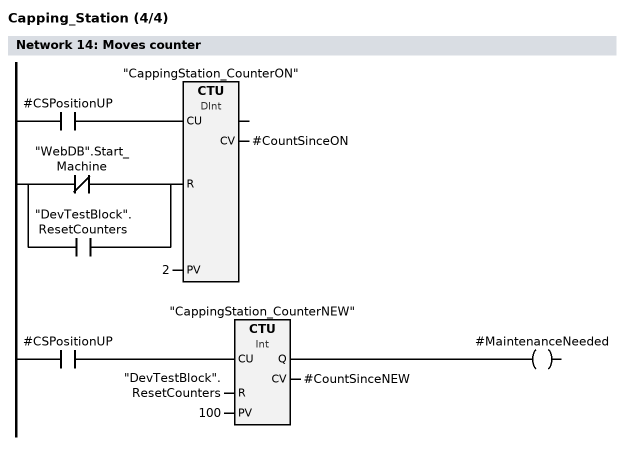
   RUNG wire#powerrail
      Contact( #CSPositionUP )
      { S7_Templates := "value_type := DInt" } "CappingStation_CounterON".CTU(r := wire#w1, pv := 2, cv => #CountSinceON)
   END_RUNG
   RUNG wire#powerrail
      I_Contact( "WebDB".Start_Machine )
   END_RUNG wire#w1
   RUNG wire#powerrail
      Contact( "DevTestBlock".ResetCounters )
   END_RUNG wire#w1
   RUNG wire#powerrail
      Contact( #CSPositionUP )
      { S7_Templates := "value_type := Int" } "CappingStation_CounterNEW".CTU(r := "DevTestBlock".ResetCounters, pv := 100, cv => #CountSinceNEW)
      Coil( #MaintenanceNeeded )
   END_RUNG
   // the same network as SCL:
   "CappingStation_CounterON".CTU(CU := #CSPositionUP,
                           R := NOT "WebDB".Start_Machine OR "DevTestBlock".ResetCounters,
                           PV := 2,
                           CV => #CountSinceON);
   "CappingStation_CounterNEW".CTU(CU := #CSPositionUP,
                           R := "DevTestBlock".ResetCounters,
                           PV := 100,
                           CV => #CountSinceNEW);
   #MaintenanceNeeded := "CappingStation_CounterNEW".Q;
END_REGION
END_FUNCTION_BLOCK

FUNCTION_BLOCK "Initial_Test_Squence"   // FB18, LAD
{ S7_Optimized_Access := 'TRUE' }
VERSION : 0.1
   VAR_INPUT
      ON : Bool;
      Position : DInt;
      HomingOK : Bool;
      InputTask : Bool;
      StepSizeInput : DInt := 100;
      AmountOfSteps : Int := 100;
   END_VAR
   VAR_OUTPUT
      StartMachine : Bool;
      StartHoming : Bool;
      StepSizeOutput : DInt := 1000;
      TestFinished : Bool;
      StartPosition : DInt;
      EndPositon : DInt;
   END_VAR
   VAR_IN_OUT
      StartTask : Bool;
   END_VAR
   VAR
      TurnOnM : Bool;
      StepNumber : Int;
      InternalWait : Bool;
      StepNumberNext : Int;
      ONM : Bool;
      TestFinishedM : Bool;
      StartTaskM : Bool;
   END_VAR
   VAR_TEMP   // added for the SCL form of the ladder/FBD networks
      _w1 : Bool;
   END_VAR
BEGIN

REGION Network 1: Turn On
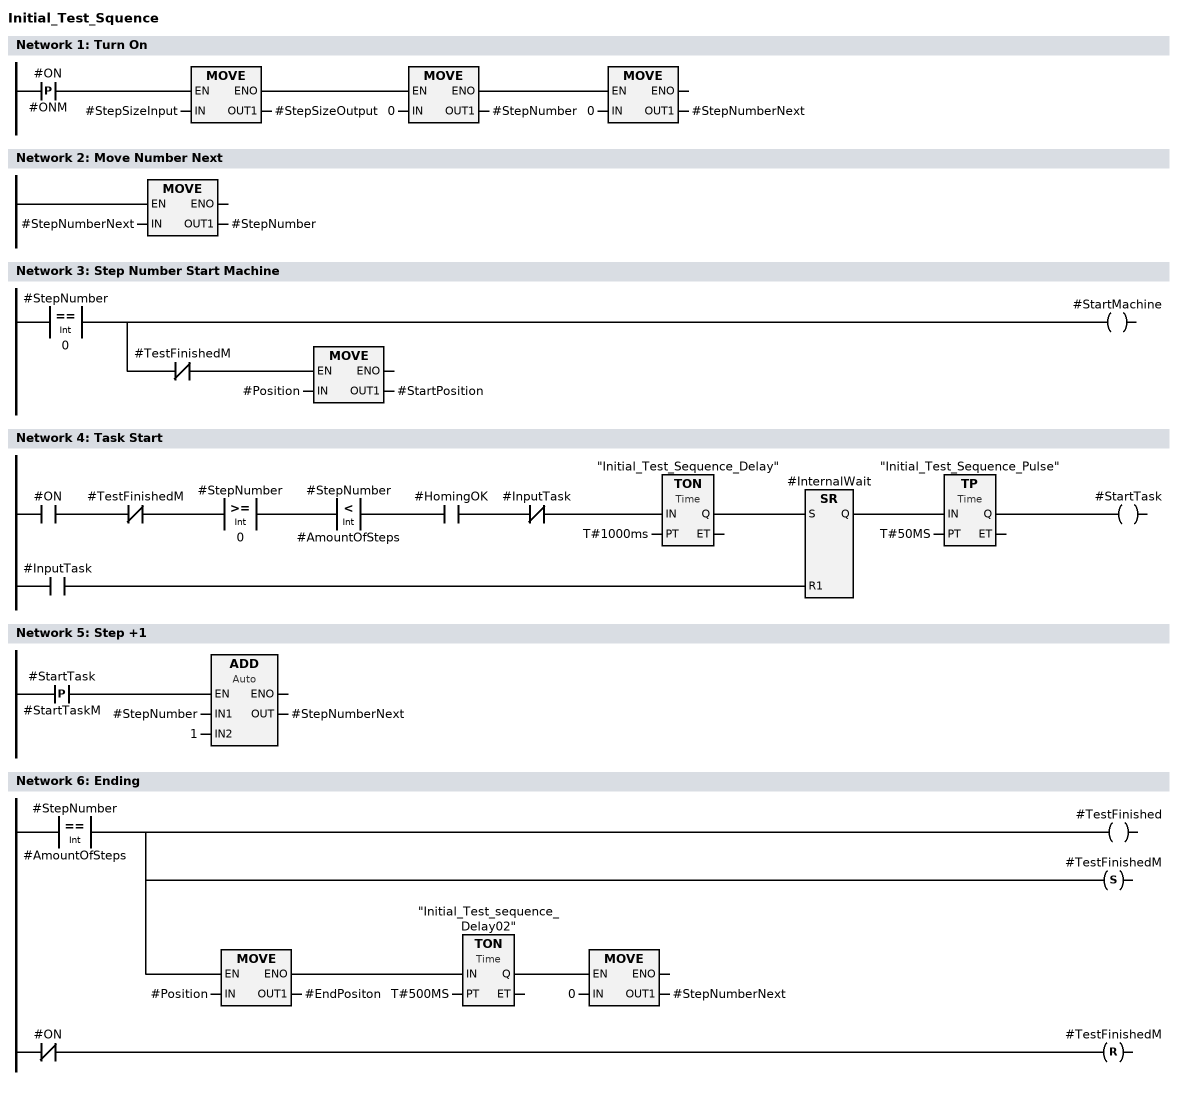
   RUNG wire#powerrail
      P_Contact(operand := #ON, bit := #ONM)
      Move(in := #StepSizeInput, out1 => #StepSizeOutput)
      Move(in := 0, out1 => #StepNumber)
      Move(in := 0, out1 => #StepNumberNext)
   END_RUNG
   // the same network as SCL:
   #_w1 := #ON AND NOT #ONM;   // rising edge of #ON
   #ONM := #ON;
   IF #_w1 THEN
       #StepSizeOutput := #StepSizeInput;
       #StepNumber := 0;
       #StepNumberNext := 0;
   END_IF;
END_REGION

REGION Network 2: Move Number Next
   RUNG wire#powerrail
      Move(in := #StepNumberNext, out1 => #StepNumber)
   END_RUNG
   // the same network as SCL:
   #StepNumber := #StepNumberNext;
END_REGION

REGION Network 3: Step Number Start Machine
   RUNG wire#powerrail
      { S7_Templates := "SrcType := Int" } EQ_Contact(in1 := #StepNumber, in2 := 0)
      wire#w1
      Coil( #StartMachine )
   END_RUNG
   RUNG wire#w1
      I_Contact( #TestFinishedM )
      Move(in := #Position, out1 => #StartPosition)
   END_RUNG
   // the same network as SCL:
   #StartMachine := #StepNumber = 0;
   IF #StartMachine AND NOT #TestFinishedM THEN #StartPosition := #Position; END_IF;
END_REGION

REGION Network 4: Task Start
   RUNG wire#powerrail
      Contact( #ON )
      I_Contact( #TestFinishedM )
      { S7_Templates := "SrcType := Int" } GE_Contact(in1 := #StepNumber, in2 := 0)
      { S7_Templates := "SrcType := Int" } LT_Contact(in1 := #StepNumber, in2 := #AmountOfSteps)
      Contact( #HomingOK )
      I_Contact( #InputTask )
      { S7_Templates := "time_type := Time" } "Initial_Test_Sequence_Delay".TON(pt := T#1000ms, et =>)
      S_SR(operand := #InternalWait, r1 := wire#w1)
      { S7_Templates := "time_type := Time" } "Initial_Test_Sequence_Pulse".TP(pt := T#50MS, et =>)
      Coil( #StartTask )
   END_RUNG
   RUNG wire#powerrail
      Contact( #InputTask )
   END_RUNG wire#w1
   // the same network as SCL:
   "Initial_Test_Sequence_Delay".TON(IN := #ON AND NOT #TestFinishedM AND (#StepNumber >= 0) AND (#StepNumber < #AmountOfSteps) AND #HomingOK AND NOT #InputTask,
                           PT := T#1000ms);
   IF "Initial_Test_Sequence_Delay".Q THEN
       #InternalWait := TRUE;   // SR flip-flop
   END_IF;
   IF #InputTask THEN #InternalWait := FALSE; END_IF;
   "Initial_Test_Sequence_Pulse".TP(IN := #InternalWait, PT := T#50MS);
   #StartTask := "Initial_Test_Sequence_Pulse".Q;
END_REGION

REGION Network 5: Step +1
   RUNG wire#powerrail
      P_Contact(operand := #StartTask, bit := #StartTaskM)
      Add(in1 := #StepNumber, in2 := 1, out => #StepNumberNext)
   END_RUNG
   // the same network as SCL:
   #_w1 := #StartTask AND NOT #StartTaskM;   // rising edge of #StartTask
   #StartTaskM := #StartTask;
   IF #_w1 THEN #StepNumberNext := #StepNumber + 1; END_IF;
END_REGION

REGION Network 6: Ending
   RUNG wire#powerrail
      { S7_Templates := "SrcType := Int" } EQ_Contact(in1 := #StepNumber, in2 := #AmountOfSteps)
      wire#w1
      Coil( #TestFinished )
   END_RUNG
   RUNG wire#w1
      S_Coil( #TestFinishedM )
   END_RUNG
   RUNG wire#w1
      Move(in := #Position, out1 => #EndPositon)
      { S7_Templates := "time_type := Time" } "Initial_Test_sequence_Delay02".TON(pt := T#500MS, et =>)
      Move(in := 0, out1 => #StepNumberNext)
   END_RUNG
   RUNG wire#powerrail
      I_Contact( #ON )
      R_Coil( #TestFinishedM )
   END_RUNG
   // the same network as SCL:
   #TestFinished := #StepNumber = #AmountOfSteps;
   IF #TestFinished THEN
       #TestFinishedM := TRUE;
       #EndPositon := #Position;
   END_IF;
   "Initial_Test_sequence_Delay02".TON(IN := #TestFinished, PT := T#500MS);
   IF "Initial_Test_sequence_Delay02".Q THEN #StepNumberNext := 0; END_IF;
   IF NOT #ON THEN #TestFinishedM := FALSE; END_IF;
END_REGION
END_FUNCTION_BLOCK

FUNCTION_BLOCK "UVLamp"   // FB19, LAD
TITLE = Description
{ S7_Optimized_Access := 'TRUE' }
VERSION : 0.1
// How to control and set the UV lamp:
// To control the lamp the machine needs to be started, all door closed and "LampFaultSignal" checked. After setting the setpoint 0-100 "LampSetpointInput" and enabling "LampEnable", the UV will work.
// 
// SafetyLimitSet - can be used to modify output range 
// 
// E-STOP - always check!
   VAR_INPUT
      Emergency : Bool;
      MachineStart : Bool;
      LampEnable : Bool;   // Device ready do use
      LampMode : Int;   // 0 by default
      LampSetpointInput : Real;   // Intensity %
      LampMaintenance : Int;   // N/A
      LampFaultSignal : Bool;   // Signal from the UV lamp
      DoorSensor : Bool;   // Connect direct
      XPosition : DInt;
      YPosition : DInt;
      WorkingRegionXstart : DInt;   // To be updated and connected to the UV lamp preferences in the MachineDB
      WorkingRegionXend : DInt := 500000;   // To be updated and connected to the UV lamp preferences in the MachineDB
      WorkingRegionYstart : DInt;   // To be updated and connected to the UV lamp preferences in the MachineDB
      WorkingRegionYend : DInt := 1500000;   // To be updated and connected to the UV lamp preferences in the MachineDB
      DevelopmentMode : Bool;
      FirstTurnOn : Bool;
   END_VAR
   VAR_OUTPUT
      LampEnabled : Bool;
      LampWorking : Bool;
      LampOutONOFF : Bool;
      LampDimming : UInt;
      LampIntensity : Real;   // Volts
      LampError : Bool;
      LampStatus : Int;   // N/A
   END_VAR
   VAR_IN_OUT
      LampInONOFF : Bool;   // Device use state
   END_VAR
   VAR
      InternalWorkingPermission : Bool;
      SetpointMax : UInt := 27648;   // 0 - 0V; 27648 - 10V;
      SetpointLimit : UInt := 27648;
      SetpointConversion : Real;
      SetpointOutput : UInt;
      SafetyLimitConversion : Real;
      IntensityConversion : Real;
   END_VAR
   VAR_TEMP
      WorkingRegionOK : Bool;
   END_VAR
   VAR CONSTANT
      SafetyLimitSet : Real := 60.0;   // 0-100%
   END_VAR
BEGIN

REGION Network 1: Working Region Check
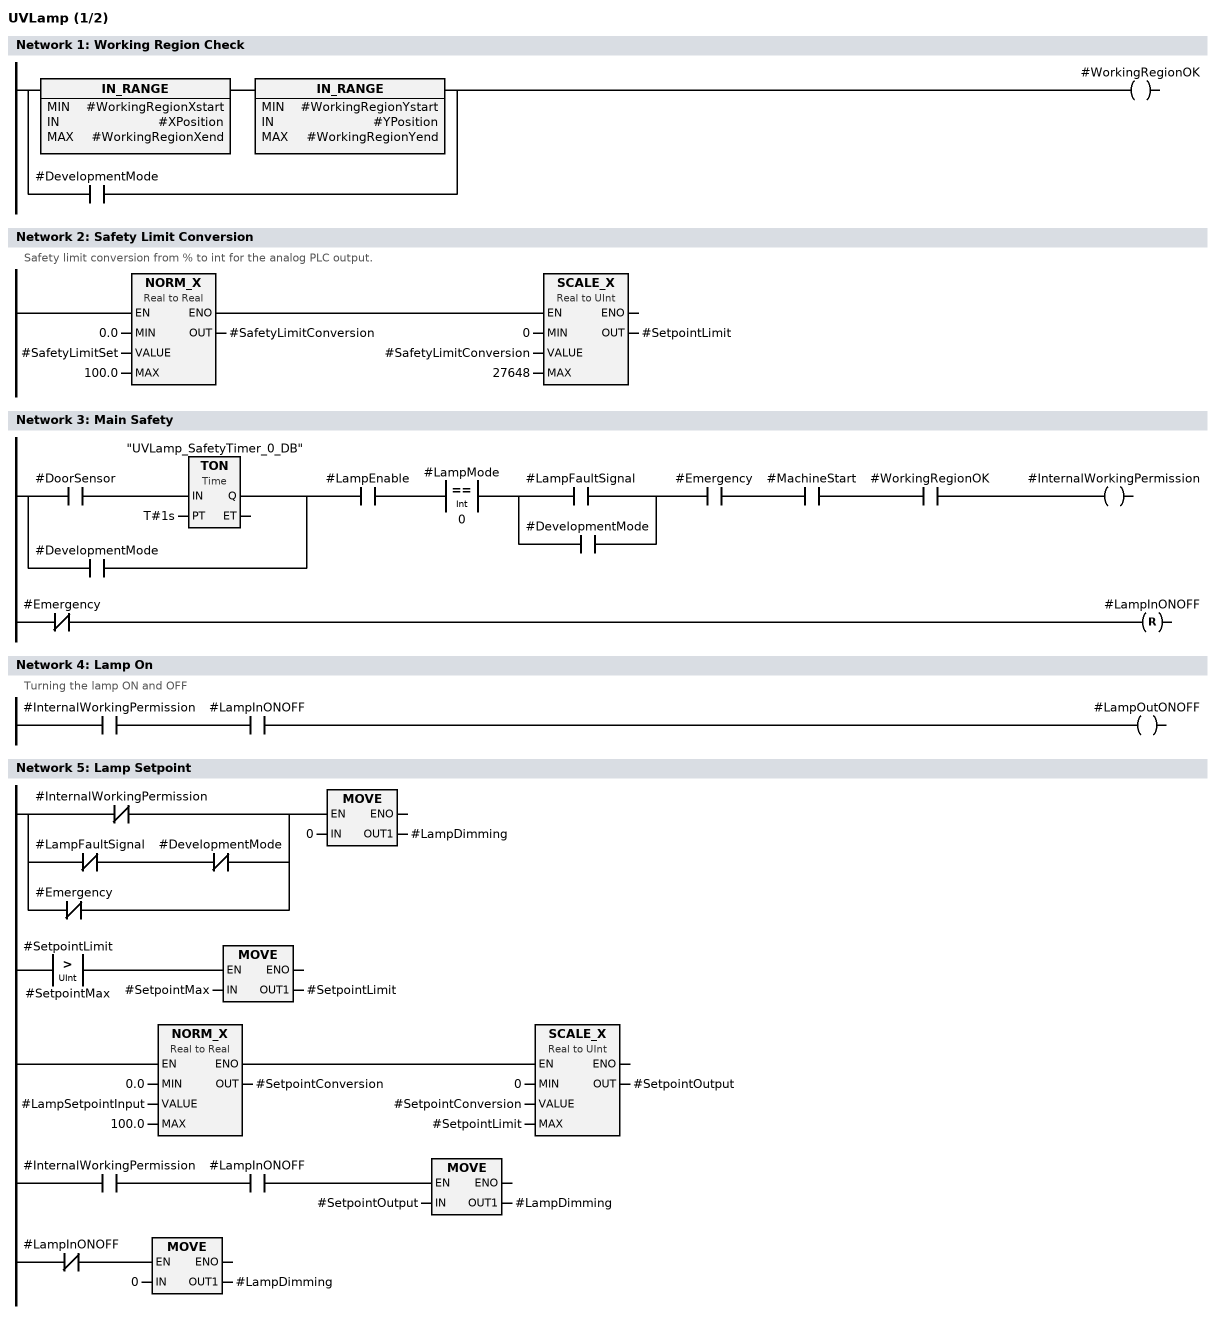
   RUNG wire#powerrail
      { S7_Templates := "SrcType := DInt" } InRange(min := #WorkingRegionXstart, in := #XPosition, max := #WorkingRegionXend)
      { S7_Templates := "SrcType := DInt" } InRange(min := #WorkingRegionYstart, in := #YPosition, max := #WorkingRegionYend)
      wire#w1
      Coil( #WorkingRegionOK )
   END_RUNG
   RUNG wire#powerrail
      Contact( #DevelopmentMode )
   END_RUNG wire#w1
   // the same network as SCL:
   #WorkingRegionOK := ((#WorkingRegionXstart <= #XPosition) AND (#XPosition <= #WorkingRegionXend) AND (#WorkingRegionYstart <= #YPosition) AND (#YPosition <= #WorkingRegionYend)) OR #DevelopmentMode;
END_REGION

REGION Network 2: Safety Limit Conversion
   // Safety limit conversion from % to int for the analog PLC output.
   RUNG wire#powerrail
      { S7_Templates := "[SrcType := Real, DestType := Real]" } Normalize(min := 0.0, value := #SafetyLimitSet, max := 100.0, out => #SafetyLimitConversion)
      { S7_Templates := "[SrcType := Real, DestType := UInt]" } Scale(min := 0, value := #SafetyLimitConversion, max := 27648, out => #SetpointLimit)
   END_RUNG
   // the same network as SCL:
   #SafetyLimitConversion := NORM_X(MIN := 0.0, VALUE := #SafetyLimitSet, MAX := 100.0);
   #SetpointLimit := SCALE_X(MIN := 0, VALUE := #SafetyLimitConversion, MAX := 27648);
END_REGION

REGION Network 3: Main Safety
   RUNG wire#powerrail
      Contact( #DoorSensor )
      { S7_Templates := "time_type := Time" } "UVLamp_SafetyTimer_0_DB".TON(pt := T#1s, et =>)
      wire#w1
      Contact( #LampEnable )
      { S7_Templates := "SrcType := Int" } EQ_Contact(in1 := #LampMode, in2 := 0)
      wire#w2
      Contact( #LampFaultSignal )
      wire#w3
      Contact( #Emergency )
      Contact( #MachineStart )
      Contact( #WorkingRegionOK )
      Coil( #InternalWorkingPermission )
   END_RUNG
   RUNG wire#powerrail
      Contact( #DevelopmentMode )
   END_RUNG wire#w1
   RUNG wire#w2
      Contact( #DevelopmentMode )
   END_RUNG wire#w3
   RUNG wire#powerrail
      I_Contact( #Emergency )
      R_Coil( #LampInONOFF )
   END_RUNG
   // the same network as SCL:
   "UVLamp_SafetyTimer_0_DB".TON(IN := #DoorSensor, PT := T#1s);
   #InternalWorkingPermission := ("UVLamp_SafetyTimer_0_DB".Q OR #DevelopmentMode) AND #LampEnable AND (#LampMode = 0) AND (#LampFaultSignal OR #DevelopmentMode) AND #Emergency AND #MachineStart AND #WorkingRegionOK;
   IF NOT #Emergency THEN #LampInONOFF := FALSE; END_IF;
END_REGION

REGION Network 4: Lamp On
   // Turning the lamp ON and OFF
   RUNG wire#powerrail
      Contact( #InternalWorkingPermission )
      Contact( #LampInONOFF )
      Coil( #LampOutONOFF )
   END_RUNG
   // the same network as SCL:
   #LampOutONOFF := #InternalWorkingPermission AND #LampInONOFF;
END_REGION

REGION Network 5: Lamp Setpoint
   RUNG wire#powerrail
      I_Contact( #InternalWorkingPermission )
      wire#w1
      Move(in := 0, out1 => #LampDimming)
   END_RUNG
   RUNG wire#powerrail
      I_Contact( #LampFaultSignal )
      I_Contact( #DevelopmentMode )
   END_RUNG wire#w1
   RUNG wire#powerrail
      I_Contact( #Emergency )
   END_RUNG wire#w1
   RUNG wire#powerrail
      { S7_Templates := "SrcType := UInt" } GT_Contact(in1 := #SetpointLimit, in2 := #SetpointMax)
      Move(in := #SetpointMax, out1 => #SetpointLimit)
   END_RUNG
   RUNG wire#powerrail
      { S7_Templates := "[SrcType := Real, DestType := Real]" } Normalize(min := 0.0, value := #LampSetpointInput, max := 100.0, out => #SetpointConversion)
      { S7_Templates := "[SrcType := Real, DestType := UInt]" } Scale(min := 0, value := #SetpointConversion, max := #SetpointLimit, out => #SetpointOutput)
   END_RUNG
   RUNG wire#powerrail
      Contact( #InternalWorkingPermission )
      Contact( #LampInONOFF )
      Move(in := #SetpointOutput, out1 => #LampDimming)
   END_RUNG
   RUNG wire#powerrail
      I_Contact( #LampInONOFF )
      Move(in := 0, out1 => #LampDimming)
   END_RUNG
   // the same network as SCL:
   IF NOT #InternalWorkingPermission OR (NOT #LampFaultSignal AND NOT #DevelopmentMode) OR NOT #Emergency THEN
       #LampDimming := 0;
   END_IF;
   IF #SetpointLimit > #SetpointMax THEN #SetpointLimit := #SetpointMax; END_IF;
   #SetpointConversion := NORM_X(MIN := 0.0, VALUE := #LampSetpointInput, MAX := 100.0);
   #SetpointOutput := SCALE_X(MIN := 0, VALUE := #SetpointConversion, MAX := #SetpointLimit);
   IF #InternalWorkingPermission AND #LampInONOFF THEN #LampDimming := #SetpointOutput; END_IF;
   IF NOT #LampInONOFF THEN #LampDimming := 0; END_IF;
END_REGION

REGION Network 6: Intensity Monitoring Conversion
   // Conversion of the intensity.
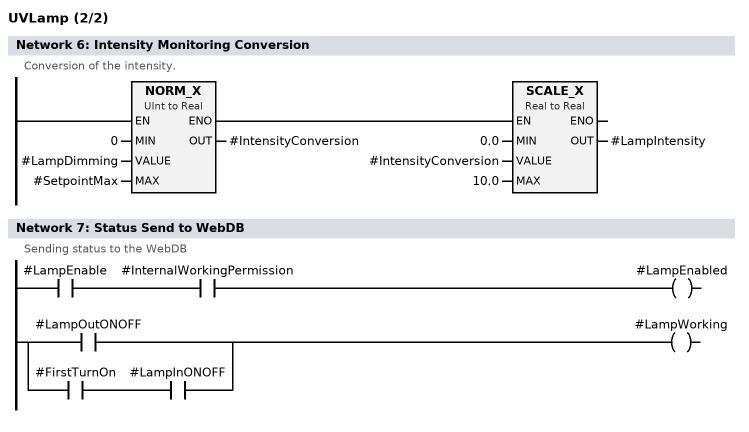
   RUNG wire#powerrail
      { S7_Templates := "[SrcType := UInt, DestType := Real]" } Normalize(min := 0, value := #LampDimming, max := #SetpointMax, out => #IntensityConversion)
      { S7_Templates := "[SrcType := Real, DestType := Real]" } Scale(min := 0.0, value := #IntensityConversion, max := 10.0, out => #LampIntensity)
   END_RUNG
   // the same network as SCL:
   #IntensityConversion := NORM_X(MIN := 0, VALUE := #LampDimming, MAX := #SetpointMax);
   #LampIntensity := SCALE_X(MIN := 0.0, VALUE := #IntensityConversion, MAX := 10.0);
END_REGION

REGION Network 7: Status Send to WebDB
   // Sending status to the WebDB
   RUNG wire#powerrail
      Contact( #LampEnable )
      Contact( #InternalWorkingPermission )
      Coil( #LampEnabled )
   END_RUNG
   RUNG wire#powerrail
      Contact( #LampOutONOFF )
      wire#w1
      Coil( #LampWorking )
   END_RUNG
   RUNG wire#powerrail
      Contact( #FirstTurnOn )
      Contact( #LampInONOFF )
   END_RUNG wire#w1
   // the same network as SCL:
   #LampEnabled := #LampEnable AND #InternalWorkingPermission;
   #LampWorking := #LampOutONOFF OR (#FirstTurnOn AND #LampInONOFF);
END_REGION
END_FUNCTION_BLOCK

FUNCTION_BLOCK "Stacklight"   // FB20, LAD
TITLE = Description:
{ S7_Optimized_Access := 'TRUE' }
VERSION : 0.1
// The stacklight is showing the status of the machine and checking different conditions:
// - errors from the drives (PLC)
// - communication (NOAH)
// - errors from the fluid supply (NOAH)
// - doors (PLC)
// 
// RED - default color, error or PLC is turning on
// ORANGE - door open or in maintenance mode
// GREEN - machine connected and working fine
// 
// RED-GREEN blinking - machine ready to connect
// 
// Date:
   VAR_INPUT
      Emergency : Bool;
      Mode : Int;
      RedIn : Bool;
      YellowIn : Bool;
      GreenIn : Bool;
      ReadyDevices : Bool;
      DoorOpen : Bool;
      Xvelocity : DInt;
      Yvelocity : DInt;
      MachineReadyPLC : Bool;
      MachineReadyNOAH : Bool;
      MachinePrintingPLC : Bool;
      MachinePrintingNOAH : Bool;
      MachineErrorPLC : Bool;
      MachineErrorNOAH : Bool;
      LED01 : Bool;
      LED02 : Bool;
      Maintenance : Int;
   END_VAR
   VAR_OUTPUT
      Status : Int;
      OutputColor : Int;
      StacklightCTRL01 : Bool;
      StacklightCTRL02 : Bool;
   END_VAR
   VAR_IN_OUT
      MachineConnectedNOAH : Bool;
   END_VAR
   VAR
      TriggerVelocityForMoving : DInt := 5;
      GreenInternal : Bool;
      YellowInternal : Bool;
      RedInternal : Bool;
      ColorInternal : Int;   // 0 = Red; 1 = Orange; 2 = Green;
      MachineMovingInternal : Bool;
      MachineConnectedPLC : Bool;
      MachineConnectedInternal : Bool;
   END_VAR
   VAR CONSTANT
      MachineConnectedWaitTime : Time := T#3s;
      MachineConnectedResetTime : Time := T#200ms;
   END_VAR
BEGIN

REGION Network 1: Machine Moving Status Read
   // Checking if the machine is moving.
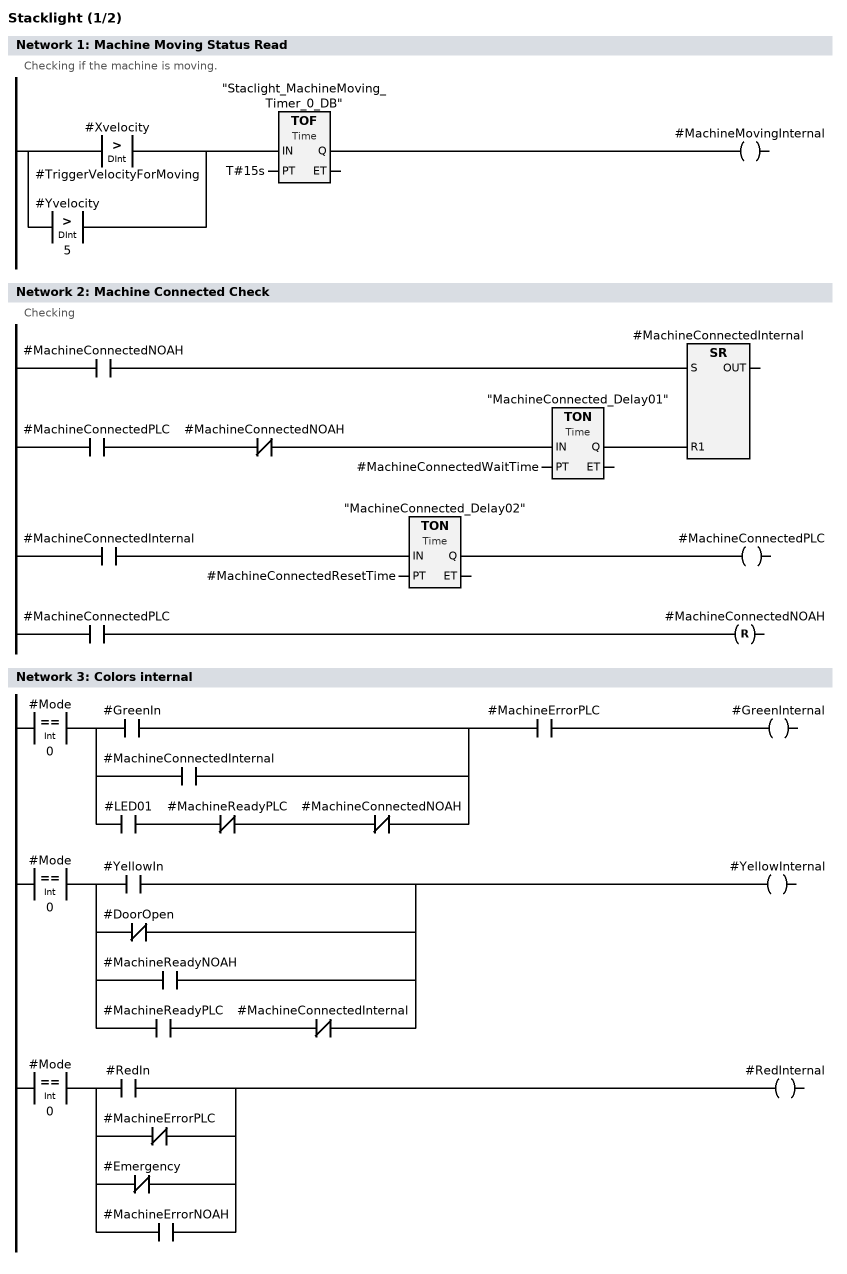
   RUNG wire#powerrail
      { S7_Templates := "SrcType := DInt" } GT_Contact(in1 := #Xvelocity, in2 := #TriggerVelocityForMoving)
      wire#w1
      { S7_Templates := "time_type := Time" } "Staclight_MachineMoving_Timer_0_DB".TOF(pt := T#15s, et =>)
      Coil( #MachineMovingInternal )
   END_RUNG
   RUNG wire#powerrail
      { S7_Templates := "SrcType := DInt" } GT_Contact(in1 := #Yvelocity, in2 := 5)
   END_RUNG wire#w1
   // the same network as SCL:
   "Staclight_MachineMoving_Timer_0_DB".TOF(IN := (#Xvelocity > #TriggerVelocityForMoving) OR (#Yvelocity > 5),
                           PT := T#15s);
   #MachineMovingInternal := "Staclight_MachineMoving_Timer_0_DB".Q;
END_REGION

REGION Network 2: Machine Connected Check
   // Checking
   RUNG wire#powerrail
      Contact( #MachineConnectedNOAH )
      S_SR(operand := #MachineConnectedInternal, r1 := wire#w1)
   END_RUNG
   RUNG wire#powerrail
      Contact( #MachineConnectedPLC )
      I_Contact( #MachineConnectedNOAH )
      { S7_Templates := "time_type := Time" } "MachineConnected_Delay01".TON(pt := #MachineConnectedWaitTime, et =>)
   END_RUNG wire#w1
   RUNG wire#powerrail
      Contact( #MachineConnectedInternal )
      { S7_Templates := "time_type := Time" } "MachineConnected_Delay02".TON(pt := #MachineConnectedResetTime, et =>)
      Coil( #MachineConnectedPLC )
   END_RUNG
   RUNG wire#powerrail
      Contact( #MachineConnectedPLC )
      R_Coil( #MachineConnectedNOAH )
   END_RUNG
   // the same network as SCL:
   "MachineConnected_Delay01".TON(IN := #MachineConnectedPLC AND NOT #MachineConnectedNOAH,
                           PT := #MachineConnectedWaitTime);
   IF #MachineConnectedNOAH THEN
       #MachineConnectedInternal := TRUE;   // SR flip-flop
   END_IF;
   IF "MachineConnected_Delay01".Q THEN #MachineConnectedInternal := FALSE; END_IF;
   "MachineConnected_Delay02".TON(IN := #MachineConnectedInternal, PT := #MachineConnectedResetTime);
   #MachineConnectedPLC := "MachineConnected_Delay02".Q;
   IF #MachineConnectedPLC THEN #MachineConnectedNOAH := FALSE; END_IF;
END_REGION

REGION Network 3: Colors internal
   RUNG wire#powerrail
      { S7_Templates := "SrcType := Int" } EQ_Contact(in1 := #Mode, in2 := 0)
      wire#w1
      Contact( #GreenIn )
      wire#w2
      Contact( #MachineErrorPLC )
      Coil( #GreenInternal )
   END_RUNG
   RUNG wire#w1
      Contact( #MachineConnectedInternal )
   END_RUNG wire#w2
   RUNG wire#w1
      Contact( #LED01 )
      I_Contact( #MachineReadyPLC )
      I_Contact( #MachineConnectedNOAH )
   END_RUNG wire#w2
   RUNG wire#powerrail
      { S7_Templates := "SrcType := Int" } EQ_Contact(in1 := #Mode, in2 := 0)
      wire#w3
      Contact( #YellowIn )
      wire#w4
      Coil( #YellowInternal )
   END_RUNG
   RUNG wire#w3
      I_Contact( #DoorOpen )
   END_RUNG wire#w4
   RUNG wire#w3
      Contact( #MachineReadyNOAH )
   END_RUNG wire#w4
   RUNG wire#w3
      Contact( #MachineReadyPLC )
      I_Contact( #MachineConnectedInternal )
   END_RUNG wire#w4
   RUNG wire#powerrail
      { S7_Templates := "SrcType := Int" } EQ_Contact(in1 := #Mode, in2 := 0)
      wire#w5
      Contact( #RedIn )
      wire#w6
      Coil( #RedInternal )
   END_RUNG
   RUNG wire#w5
      I_Contact( #MachineErrorPLC )
   END_RUNG wire#w6
   RUNG wire#w5
      I_Contact( #Emergency )
   END_RUNG wire#w6
   RUNG wire#w5
      Contact( #MachineErrorNOAH )
   END_RUNG wire#w6
   // the same network as SCL:
   #GreenInternal := (#Mode = 0) AND (#GreenIn OR #MachineConnectedInternal OR (#LED01 AND NOT #MachineReadyPLC AND NOT #MachineConnectedNOAH)) AND #MachineErrorPLC;
   #YellowInternal := (#Mode = 0) AND (#YellowIn OR NOT #DoorOpen OR #MachineReadyNOAH OR (#MachineReadyPLC AND NOT #MachineConnectedInternal));
   #RedInternal := (#Mode = 0) AND (#RedIn OR NOT #MachineErrorPLC OR NOT #Emergency OR #MachineErrorNOAH);
END_REGION

REGION Network 4: Status Move
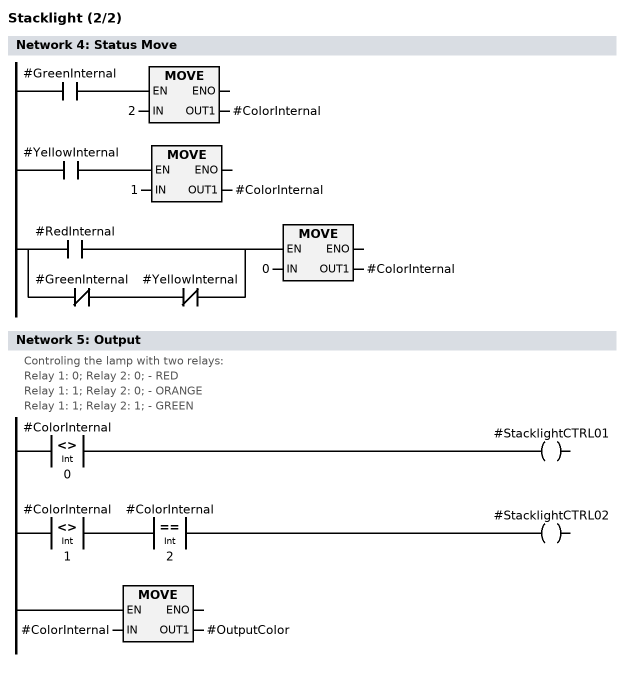
   RUNG wire#powerrail
      Contact( #GreenInternal )
      Move(in := 2, out1 => #ColorInternal)
   END_RUNG
   RUNG wire#powerrail
      Contact( #YellowInternal )
      Move(in := 1, out1 => #ColorInternal)
   END_RUNG
   RUNG wire#powerrail
      Contact( #RedInternal )
      wire#w1
      Move(in := 0, out1 => #ColorInternal)
   END_RUNG
   RUNG wire#powerrail
      I_Contact( #GreenInternal )
      I_Contact( #YellowInternal )
   END_RUNG wire#w1
   // the same network as SCL:
   IF #GreenInternal THEN #ColorInternal := 2; END_IF;
   IF #YellowInternal THEN #ColorInternal := 1; END_IF;
   IF #RedInternal OR (NOT #GreenInternal AND NOT #YellowInternal) THEN #ColorInternal := 0; END_IF;
END_REGION

REGION Network 5: Output
   // Controling the lamp with two relays:
   // Relay 1: 0; Relay 2: 0; - RED
   // Relay 1: 1; Relay 2: 0; - ORANGE
   // Relay 1: 1; Relay 2: 1; - GREEN
   RUNG wire#powerrail
      { S7_Templates := "SrcType := Int" } NE_Contact(in1 := #ColorInternal, in2 := 0)
      Coil( #StacklightCTRL01 )
   END_RUNG
   RUNG wire#powerrail
      { S7_Templates := "SrcType := Int" } NE_Contact(in1 := #ColorInternal, in2 := 1)
      { S7_Templates := "SrcType := Int" } EQ_Contact(in1 := #ColorInternal, in2 := 2)
      Coil( #StacklightCTRL02 )
   END_RUNG
   RUNG wire#powerrail
      Move(in := #ColorInternal, out1 => #OutputColor)
   END_RUNG
   // the same network as SCL:
   #StacklightCTRL01 := #ColorInternal <> 0;
   #StacklightCTRL02 := (#ColorInternal <> 1) AND (#ColorInternal = 2);
   #OutputColor := #ColorInternal;
END_REGION
END_FUNCTION_BLOCK

FUNCTION_BLOCK "Control_Buttons_Activation"   // FB23, LAD
{ S7_Optimized_Access := 'TRUE' }
VERSION : 0.1
   VAR_INPUT
      JogInZ1pos : Bool;
      JogInZ1neg : Bool;
      JogInZ2pos : Bool;
      JogInZ2neg : Bool;
   END_VAR
   VAR_OUTPUT
      Control_Buttons_Move_Permission : Bool;
      Control_Buttons_ActivatedOUT : Bool;
   END_VAR
   VAR
      Step01 : Bool;
      Step02 : Bool;
      Step03 : Bool;
      Step04 : Bool;
      Step05 : Bool;
      Step06 : Bool;
      Step07 : Bool;
      Step08 : Bool;
      AnyButtonPressed : Bool;
      AllButtonsPressed : Bool;
      ControlButtonsActivated : Bool;
   END_VAR
BEGIN

REGION Network 1: Any Button Pressed
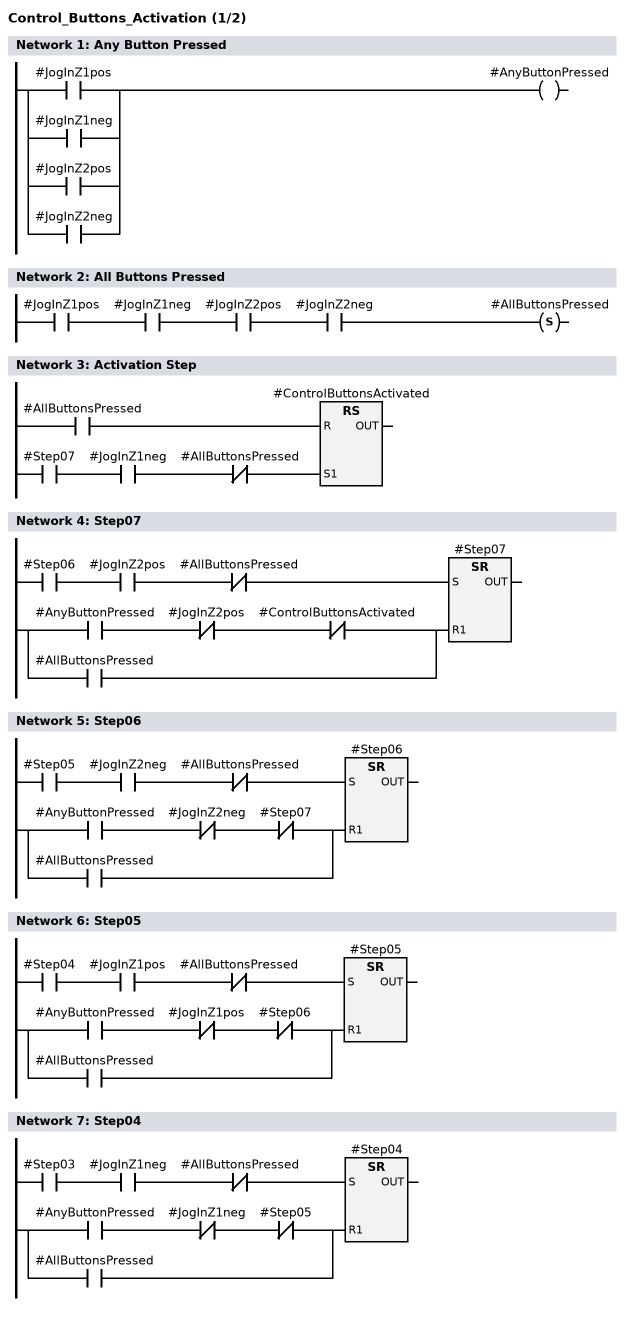
   RUNG wire#powerrail
      Contact( #JogInZ1pos )
      wire#w1
      Coil( #AnyButtonPressed )
   END_RUNG
   RUNG wire#powerrail
      Contact( #JogInZ1neg )
   END_RUNG wire#w1
   RUNG wire#powerrail
      Contact( #JogInZ2pos )
   END_RUNG wire#w1
   RUNG wire#powerrail
      Contact( #JogInZ2neg )
   END_RUNG wire#w1
   // the same network as SCL:
   #AnyButtonPressed := #JogInZ1pos OR #JogInZ1neg OR #JogInZ2pos OR #JogInZ2neg;
END_REGION

REGION Network 2: All Buttons Pressed
   RUNG wire#powerrail
      Contact( #JogInZ1pos )
      Contact( #JogInZ1neg )
      Contact( #JogInZ2pos )
      Contact( #JogInZ2neg )
      S_Coil( #AllButtonsPressed )
   END_RUNG
   // the same network as SCL:
   IF #JogInZ1pos AND #JogInZ1neg AND #JogInZ2pos AND #JogInZ2neg THEN #AllButtonsPressed := TRUE; END_IF;
END_REGION

REGION Network 3: Activation Step
   RUNG wire#powerrail
      Contact( #AllButtonsPressed )
      S_RS(operand := #ControlButtonsActivated, s1 := wire#w1)
   END_RUNG
   RUNG wire#powerrail
      Contact( #Step07 )
      Contact( #JogInZ1neg )
      I_Contact( #AllButtonsPressed )
   END_RUNG wire#w1
   // the same network as SCL:
   IF #AllButtonsPressed THEN
       #ControlButtonsActivated := FALSE;   // RS flip-flop
   END_IF;
   IF #Step07 AND #JogInZ1neg AND NOT #AllButtonsPressed THEN #ControlButtonsActivated := TRUE; END_IF;
END_REGION

REGION Network 4: Step07
   RUNG wire#powerrail
      Contact( #Step06 )
      Contact( #JogInZ2pos )
      I_Contact( #AllButtonsPressed )
      S_SR(operand := #Step07, r1 := wire#w1)
   END_RUNG
   RUNG wire#powerrail
      Contact( #AnyButtonPressed )
      I_Contact( #JogInZ2pos )
      I_Contact( #ControlButtonsActivated )
   END_RUNG wire#w1
   RUNG wire#powerrail
      Contact( #AllButtonsPressed )
   END_RUNG wire#w1
   // the same network as SCL:
   IF #Step06 AND #JogInZ2pos AND NOT #AllButtonsPressed THEN
       #Step07 := TRUE;   // SR flip-flop
   END_IF;
   IF (#AnyButtonPressed AND NOT #JogInZ2pos AND NOT #ControlButtonsActivated) OR #AllButtonsPressed THEN
       #Step07 := FALSE;
   END_IF;
END_REGION

REGION Network 5: Step06
   RUNG wire#powerrail
      Contact( #Step05 )
      Contact( #JogInZ2neg )
      I_Contact( #AllButtonsPressed )
      S_SR(operand := #Step06, r1 := wire#w1)
   END_RUNG
   RUNG wire#powerrail
      Contact( #AnyButtonPressed )
      I_Contact( #JogInZ2neg )
      I_Contact( #Step07 )
   END_RUNG wire#w1
   RUNG wire#powerrail
      Contact( #AllButtonsPressed )
   END_RUNG wire#w1
   // the same network as SCL:
   IF #Step05 AND #JogInZ2neg AND NOT #AllButtonsPressed THEN
       #Step06 := TRUE;   // SR flip-flop
   END_IF;
   IF (#AnyButtonPressed AND NOT #JogInZ2neg AND NOT #Step07) OR #AllButtonsPressed THEN
       #Step06 := FALSE;
   END_IF;
END_REGION

REGION Network 6: Step05
   RUNG wire#powerrail
      Contact( #Step04 )
      Contact( #JogInZ1pos )
      I_Contact( #AllButtonsPressed )
      S_SR(operand := #Step05, r1 := wire#w1)
   END_RUNG
   RUNG wire#powerrail
      Contact( #AnyButtonPressed )
      I_Contact( #JogInZ1pos )
      I_Contact( #Step06 )
   END_RUNG wire#w1
   RUNG wire#powerrail
      Contact( #AllButtonsPressed )
   END_RUNG wire#w1
   // the same network as SCL:
   IF #Step04 AND #JogInZ1pos AND NOT #AllButtonsPressed THEN
       #Step05 := TRUE;   // SR flip-flop
   END_IF;
   IF (#AnyButtonPressed AND NOT #JogInZ1pos AND NOT #Step06) OR #AllButtonsPressed THEN
       #Step05 := FALSE;
   END_IF;
END_REGION

REGION Network 7: Step04
   RUNG wire#powerrail
      Contact( #Step03 )
      Contact( #JogInZ1neg )
      I_Contact( #AllButtonsPressed )
      S_SR(operand := #Step04, r1 := wire#w1)
   END_RUNG
   RUNG wire#powerrail
      Contact( #AnyButtonPressed )
      I_Contact( #JogInZ1neg )
      I_Contact( #Step05 )
   END_RUNG wire#w1
   RUNG wire#powerrail
      Contact( #AllButtonsPressed )
   END_RUNG wire#w1
   // the same network as SCL:
   IF #Step03 AND #JogInZ1neg AND NOT #AllButtonsPressed THEN
       #Step04 := TRUE;   // SR flip-flop
   END_IF;
   IF (#AnyButtonPressed AND NOT #JogInZ1neg AND NOT #Step05) OR #AllButtonsPressed THEN
       #Step04 := FALSE;
   END_IF;
END_REGION

REGION Network 8: Step03
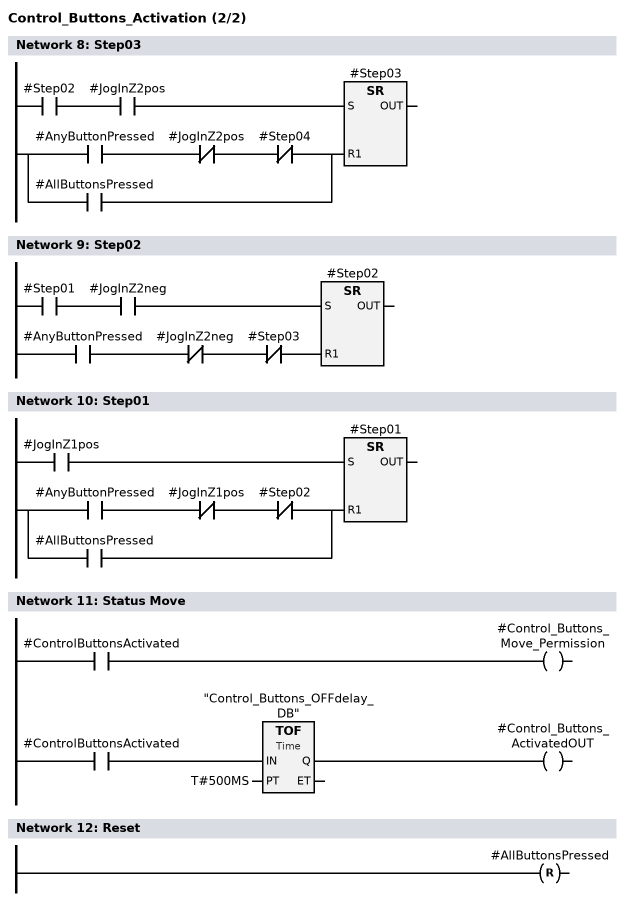
   RUNG wire#powerrail
      Contact( #Step02 )
      Contact( #JogInZ2pos )
      S_SR(operand := #Step03, r1 := wire#w1)
   END_RUNG
   RUNG wire#powerrail
      Contact( #AnyButtonPressed )
      I_Contact( #JogInZ2pos )
      I_Contact( #Step04 )
   END_RUNG wire#w1
   RUNG wire#powerrail
      Contact( #AllButtonsPressed )
   END_RUNG wire#w1
   // the same network as SCL:
   IF #Step02 AND #JogInZ2pos THEN
       #Step03 := TRUE;   // SR flip-flop
   END_IF;
   IF (#AnyButtonPressed AND NOT #JogInZ2pos AND NOT #Step04) OR #AllButtonsPressed THEN
       #Step03 := FALSE;
   END_IF;
END_REGION

REGION Network 9: Step02
   RUNG wire#powerrail
      Contact( #Step01 )
      Contact( #JogInZ2neg )
      S_SR(operand := #Step02, r1 := wire#w1)
   END_RUNG
   RUNG wire#powerrail
      Contact( #AnyButtonPressed )
      I_Contact( #JogInZ2neg )
      I_Contact( #Step03 )
   END_RUNG wire#w1
   // the same network as SCL:
   IF #Step01 AND #JogInZ2neg THEN
       #Step02 := TRUE;   // SR flip-flop
   END_IF;
   IF #AnyButtonPressed AND NOT #JogInZ2neg AND NOT #Step03 THEN #Step02 := FALSE; END_IF;
END_REGION

REGION Network 10: Step01
   RUNG wire#powerrail
      Contact( #JogInZ1pos )
      S_SR(operand := #Step01, r1 := wire#w1)
   END_RUNG
   RUNG wire#powerrail
      Contact( #AnyButtonPressed )
      I_Contact( #JogInZ1pos )
      I_Contact( #Step02 )
   END_RUNG wire#w1
   RUNG wire#powerrail
      Contact( #AllButtonsPressed )
   END_RUNG wire#w1
   // the same network as SCL:
   IF #JogInZ1pos THEN
       #Step01 := TRUE;   // SR flip-flop
   END_IF;
   IF (#AnyButtonPressed AND NOT #JogInZ1pos AND NOT #Step02) OR #AllButtonsPressed THEN
       #Step01 := FALSE;
   END_IF;
END_REGION

REGION Network 11: Status Move
   RUNG wire#powerrail
      Contact( #ControlButtonsActivated )
      Coil( #Control_Buttons_Move_Permission )
   END_RUNG
   RUNG wire#powerrail
      Contact( #ControlButtonsActivated )
      { S7_Templates := "time_type := Time" } "Control_Buttons_OFFdelay_DB".TOF(pt := T#500MS, et =>)
      Coil( #Control_Buttons_ActivatedOUT )
   END_RUNG
   // the same network as SCL:
   #Control_Buttons_Move_Permission := #ControlButtonsActivated;
   "Control_Buttons_OFFdelay_DB".TOF(IN := #ControlButtonsActivated, PT := T#500MS);
   #Control_Buttons_ActivatedOUT := "Control_Buttons_OFFdelay_DB".Q;
END_REGION

REGION Network 12: Reset
   RUNG wire#powerrail
      R_Coil( #AllButtonsPressed )
   END_RUNG
   // the same network as SCL:
   #AllButtonsPressed := FALSE;
END_REGION
END_FUNCTION_BLOCK

FUNCTION_BLOCK "Control_Buttons_Manipulate"   // FB24, LAD
{ S7_Optimized_Access := 'TRUE' }
VERSION : 0.1
// Simple control block to activate printhead motion in X and Y direction
   VAR_INPUT
      JogInZ1pos : Bool;
      JogInZ1neg : Bool;
      JogInZ2pos : Bool;
      JogInZ2neg : Bool;
      InXhome : Bool;
      InYhome : Bool;
      InZ1home : Bool;
      InZ2home : Bool;
      MovePermission : Bool;
      ReadyDevices : Bool;
   END_VAR
   VAR_OUTPUT
      JogOutXpos : Bool;
      JogOutXneg : Bool;
      JogOutYpos : Bool;
      JogOutYneg : Bool;
      JogOutZ1pos : Bool;
      JogOutZ1neg : Bool;
      JogOutZ2pos : Bool;
      JogOutZ2neg : Bool;
      XHoming : Bool;
      YHoming : Bool;
      Z1Homing : Bool;
      Z2Homing : Bool;
      StartMachine : Bool;
   END_VAR
   VAR
      ButtonsReadyToRead : Bool;
      XYmoveout : Bool;
   END_VAR
BEGIN

REGION Network 1: Start Machine
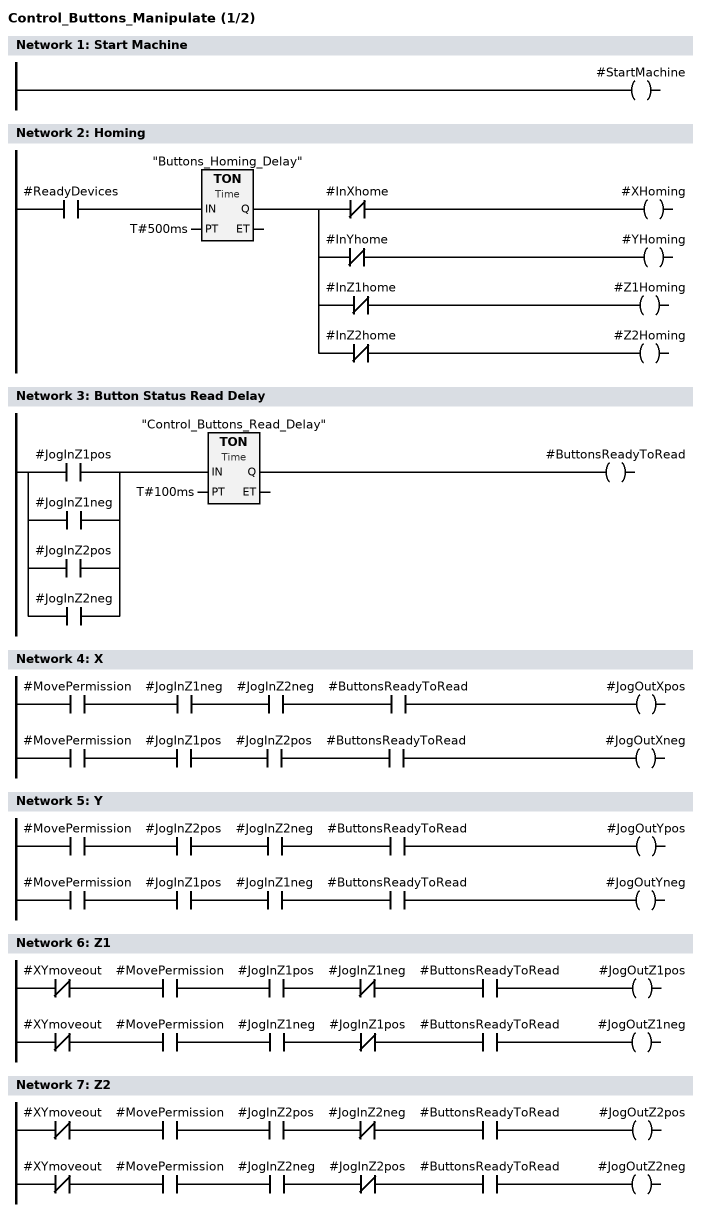
   RUNG wire#powerrail
      Coil( #StartMachine )
   END_RUNG
   // the same network as SCL:
   #StartMachine := TRUE;
END_REGION

REGION Network 2: Homing
   RUNG wire#powerrail
      Contact( #ReadyDevices )
      { S7_Templates := "time_type := Time" } "Buttons_Homing_Delay".TON(pt := T#500ms, et =>)
      wire#w1
      I_Contact( #InXhome )
      Coil( #XHoming )
   END_RUNG
   RUNG wire#w1
      I_Contact( #InYhome )
      Coil( #YHoming )
   END_RUNG
   RUNG wire#w1
      I_Contact( #InZ1home )
      Coil( #Z1Homing )
   END_RUNG
   RUNG wire#w1
      I_Contact( #InZ2home )
      Coil( #Z2Homing )
   END_RUNG
   // the same network as SCL:
   "Buttons_Homing_Delay".TON(IN := #ReadyDevices, PT := T#500ms);
   #XHoming := "Buttons_Homing_Delay".Q AND NOT #InXhome;
   #YHoming := "Buttons_Homing_Delay".Q AND NOT #InYhome;
   #Z1Homing := "Buttons_Homing_Delay".Q AND NOT #InZ1home;
   #Z2Homing := "Buttons_Homing_Delay".Q AND NOT #InZ2home;
END_REGION

REGION Network 3: Button Status Read Delay
   RUNG wire#powerrail
      Contact( #JogInZ1pos )
      wire#w1
      { S7_Templates := "time_type := Time" } "Control_Buttons_Read_Delay".TON(pt := T#100ms, et =>)
      Coil( #ButtonsReadyToRead )
   END_RUNG
   RUNG wire#powerrail
      Contact( #JogInZ1neg )
   END_RUNG wire#w1
   RUNG wire#powerrail
      Contact( #JogInZ2pos )
   END_RUNG wire#w1
   RUNG wire#powerrail
      Contact( #JogInZ2neg )
   END_RUNG wire#w1
   // the same network as SCL:
   "Control_Buttons_Read_Delay".TON(IN := #JogInZ1pos OR #JogInZ1neg OR #JogInZ2pos OR #JogInZ2neg,
                           PT := T#100ms);
   #ButtonsReadyToRead := "Control_Buttons_Read_Delay".Q;
END_REGION

REGION Network 4: X
   RUNG wire#powerrail
      Contact( #MovePermission )
      Contact( #JogInZ1neg )
      Contact( #JogInZ2neg )
      Contact( #ButtonsReadyToRead )
      Coil( #JogOutXpos )
   END_RUNG
   RUNG wire#powerrail
      Contact( #MovePermission )
      Contact( #JogInZ1pos )
      Contact( #JogInZ2pos )
      Contact( #ButtonsReadyToRead )
      Coil( #JogOutXneg )
   END_RUNG
   // the same network as SCL:
   #JogOutXpos := #MovePermission AND #JogInZ1neg AND #JogInZ2neg AND #ButtonsReadyToRead;
   #JogOutXneg := #MovePermission AND #JogInZ1pos AND #JogInZ2pos AND #ButtonsReadyToRead;
END_REGION

REGION Network 5: Y
   RUNG wire#powerrail
      Contact( #MovePermission )
      Contact( #JogInZ2pos )
      Contact( #JogInZ2neg )
      Contact( #ButtonsReadyToRead )
      Coil( #JogOutYpos )
   END_RUNG
   RUNG wire#powerrail
      Contact( #MovePermission )
      Contact( #JogInZ1pos )
      Contact( #JogInZ1neg )
      Contact( #ButtonsReadyToRead )
      Coil( #JogOutYneg )
   END_RUNG
   // the same network as SCL:
   #JogOutYpos := #MovePermission AND #JogInZ2pos AND #JogInZ2neg AND #ButtonsReadyToRead;
   #JogOutYneg := #MovePermission AND #JogInZ1pos AND #JogInZ1neg AND #ButtonsReadyToRead;
END_REGION

REGION Network 6: Z1
   RUNG wire#powerrail
      I_Contact( #XYmoveout )
      Contact( #MovePermission )
      Contact( #JogInZ1pos )
      I_Contact( #JogInZ1neg )
      Contact( #ButtonsReadyToRead )
      Coil( #JogOutZ1pos )
   END_RUNG
   RUNG wire#powerrail
      I_Contact( #XYmoveout )
      Contact( #MovePermission )
      Contact( #JogInZ1neg )
      I_Contact( #JogInZ1pos )
      Contact( #ButtonsReadyToRead )
      Coil( #JogOutZ1neg )
   END_RUNG
   // the same network as SCL:
   #JogOutZ1pos := NOT #XYmoveout AND #MovePermission AND #JogInZ1pos AND NOT #JogInZ1neg AND #ButtonsReadyToRead;
   #JogOutZ1neg := NOT #XYmoveout AND #MovePermission AND #JogInZ1neg AND NOT #JogInZ1pos AND #ButtonsReadyToRead;
END_REGION

REGION Network 7: Z2
   RUNG wire#powerrail
      I_Contact( #XYmoveout )
      Contact( #MovePermission )
      Contact( #JogInZ2pos )
      I_Contact( #JogInZ2neg )
      Contact( #ButtonsReadyToRead )
      Coil( #JogOutZ2pos )
   END_RUNG
   RUNG wire#powerrail
      I_Contact( #XYmoveout )
      Contact( #MovePermission )
      Contact( #JogInZ2neg )
      I_Contact( #JogInZ2pos )
      Contact( #ButtonsReadyToRead )
      Coil( #JogOutZ2neg )
   END_RUNG
   // the same network as SCL:
   #JogOutZ2pos := NOT #XYmoveout AND #MovePermission AND #JogInZ2pos AND NOT #JogInZ2neg AND #ButtonsReadyToRead;
   #JogOutZ2neg := NOT #XYmoveout AND #MovePermission AND #JogInZ2neg AND NOT #JogInZ2pos AND #ButtonsReadyToRead;
END_REGION

REGION Network 8: Status
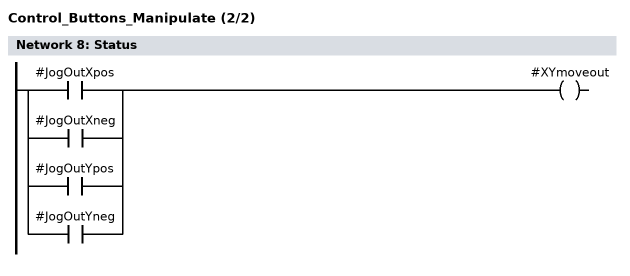
   RUNG wire#powerrail
      Contact( #JogOutXpos )
      wire#w1
      Coil( #XYmoveout )
   END_RUNG
   RUNG wire#powerrail
      Contact( #JogOutXneg )
   END_RUNG wire#w1
   RUNG wire#powerrail
      Contact( #JogOutYpos )
   END_RUNG wire#w1
   RUNG wire#powerrail
      Contact( #JogOutYneg )
   END_RUNG wire#w1
   // the same network as SCL:
   #XYmoveout := #JogOutXpos OR #JogOutXneg OR #JogOutYpos OR #JogOutYneg;
END_REGION
END_FUNCTION_BLOCK

FUNCTION_BLOCK "DataLogging"   // FB4, LAD
{ S7_Optimized_Access := 'TRUE' }
VERSION : 0.1
   VAR_INPUT
      CreateFile : Bool;
      StartLogging : Bool;
      Variable01in_Bool : Bool;
      Name_01 : String;
      Variable02in_Bool : Bool;
      Name_02 : String;
      Variable03in_Dint : DInt;
      Name_03 : String;
      Variable04in_Dint : DInt;
      Name_04 : String;
      Variable05in_Dint : DInt;
      Name_05 : String;
      Variable06in_Dint : DInt;
      Name_06 : String;
   END_VAR
   VAR_OUTPUT
      Variable01out_Bool : Bool;
      Variable02out_Bool : Bool;
      Variable03out_Dint : DInt;
      Variable04out_Dint : DInt;
      Variable05out_Dint : DInt;
      Variable06out_Dint : DInt;
      LogColumns : String;
   END_VAR
   VAR
      FileName : String := 'Logging_Test_01';
      REQ : Bool;
      ID : DWord;
      StartingTime : DTL;
      ReturnValue : Int;
      AmountOfRecords : UDInt := 10000;   // For 864000 and 10 records per sec = 24h
      StartLoggingM : Bool;
      WriteColumn : Int;
      Column01Internal : String;
      Column02Internal : String;
      Column03Internal : String;
      Column04Internal : String;
      Column05Internal : String;
      Column06Internal : String;
      WriteColumnReady : Bool;
      RecordCount : DInt;
   END_VAR
   VAR CONSTANT
      NameOfColumn01 : String := 'TestColumn_01';
      NameOfColumn02 : String := 'TestColumn_02';
   END_VAR
   VAR_TEMP   // added for the SCL form of the ladder/FBD networks
      _w1 : Bool;
      _w2 : Bool;
      _w3 : Bool;
      _w4 : Bool;
      _w5 : Bool;
   END_VAR
BEGIN

REGION Network 1: Start logging
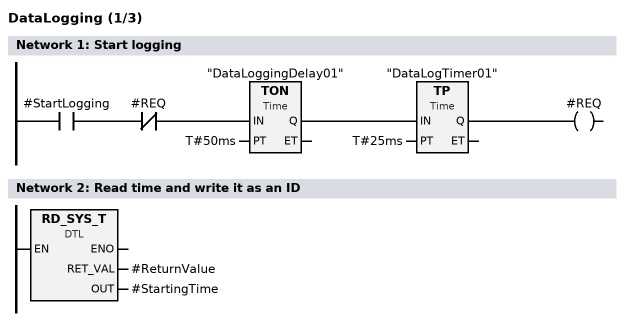
   RUNG wire#powerrail
      Contact( #StartLogging )
      I_Contact( #REQ )
      { S7_Templates := "time_type := Time" } "DataLoggingDelay01".TON(pt := T#50ms, et =>)
      { S7_Templates := "time_type := Time" } "DataLogTimer01".TP(pt := T#25ms, et =>)
      Coil( #REQ )
   END_RUNG
   // the same network as SCL:
   "DataLoggingDelay01".TON(IN := #StartLogging AND NOT #REQ, PT := T#50ms);
   "DataLogTimer01".TP(IN := "DataLoggingDelay01".Q, PT := T#25ms);
   #REQ := "DataLogTimer01".Q;
END_REGION

REGION Network 2: Read time and write it as an ID
   RUNG wire#powerrail
      { S7_Templates := "date_type := DTL" } RD_SYS_T(RET_VAL => #ReturnValue, OUT => #StartingTime)
   END_RUNG
   // the same network as SCL:
   #ReturnValue := RD_SYS_T(OUT => #StartingTime);
END_REGION

REGION Network 3: Write Column Names
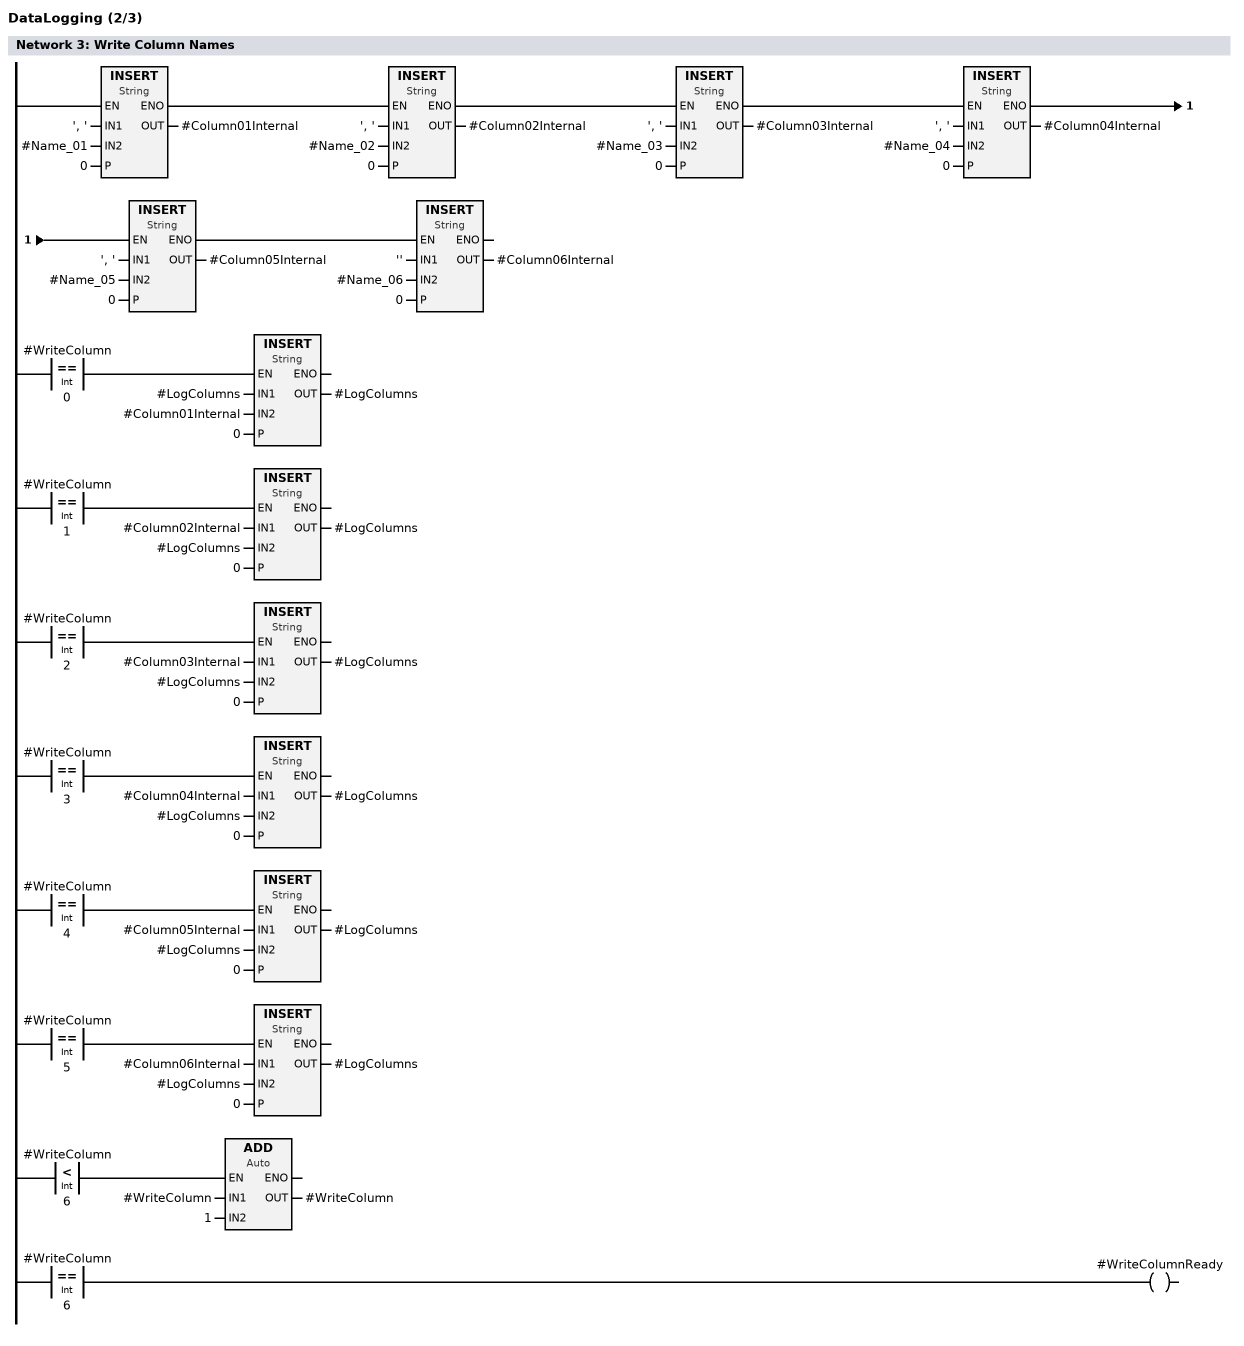
   RUNG wire#powerrail
      { S7_Templates := "str_type := String" } INSERT(IN1 := ', ', IN2 := #Name_01, P := 0, OUT => #Column01Internal)
      { S7_Templates := "str_type := String" } INSERT(IN1 := ', ', IN2 := #Name_02, P := 0, OUT => #Column02Internal)
      { S7_Templates := "str_type := String" } INSERT(IN1 := ', ', IN2 := #Name_03, P := 0, OUT => #Column03Internal)
      { S7_Templates := "str_type := String" } INSERT(IN1 := ', ', IN2 := #Name_04, P := 0, OUT => #Column04Internal)
      { S7_Templates := "str_type := String" } INSERT(IN1 := ', ', IN2 := #Name_05, P := 0, OUT => #Column05Internal)
      { S7_Templates := "str_type := String" } INSERT(IN1 := '', IN2 := #Name_06, P := 0, OUT => #Column06Internal)
   END_RUNG
   RUNG wire#powerrail
      { S7_Templates := "SrcType := Int" } EQ_Contact(in1 := #WriteColumn, in2 := 0)
      { S7_Templates := "str_type := String" } INSERT(IN1 := #LogColumns, IN2 := #Column01Internal, P := 0, OUT => #LogColumns)
   END_RUNG
   RUNG wire#powerrail
      { S7_Templates := "SrcType := Int" } EQ_Contact(in1 := #WriteColumn, in2 := 1)
      { S7_Templates := "str_type := String" } INSERT(IN1 := #Column02Internal, IN2 := #LogColumns, P := 0, OUT => #LogColumns)
   END_RUNG
   RUNG wire#powerrail
      { S7_Templates := "SrcType := Int" } EQ_Contact(in1 := #WriteColumn, in2 := 2)
      { S7_Templates := "str_type := String" } INSERT(IN1 := #Column03Internal, IN2 := #LogColumns, P := 0, OUT => #LogColumns)
   END_RUNG
   RUNG wire#powerrail
      { S7_Templates := "SrcType := Int" } EQ_Contact(in1 := #WriteColumn, in2 := 3)
      { S7_Templates := "str_type := String" } INSERT(IN1 := #Column04Internal, IN2 := #LogColumns, P := 0, OUT => #LogColumns)
   END_RUNG
   RUNG wire#powerrail
      { S7_Templates := "SrcType := Int" } EQ_Contact(in1 := #WriteColumn, in2 := 4)
      { S7_Templates := "str_type := String" } INSERT(IN1 := #Column05Internal, IN2 := #LogColumns, P := 0, OUT => #LogColumns)
   END_RUNG
   RUNG wire#powerrail
      { S7_Templates := "SrcType := Int" } EQ_Contact(in1 := #WriteColumn, in2 := 5)
      { S7_Templates := "str_type := String" } INSERT(IN1 := #Column06Internal, IN2 := #LogColumns, P := 0, OUT => #LogColumns)
   END_RUNG
   RUNG wire#powerrail
      { S7_Templates := "SrcType := Int" } LT_Contact(in1 := #WriteColumn, in2 := 6)
      Add(in1 := #WriteColumn, in2 := 1, out => #WriteColumn)
   END_RUNG
   RUNG wire#powerrail
      { S7_Templates := "SrcType := Int" } EQ_Contact(in1 := #WriteColumn, in2 := 6)
      Coil( #WriteColumnReady )
   END_RUNG
   // the same network as SCL:
   INSERT(IN1 := ', ', IN2 := #Name_01, P := 0, OUT => #Column01Internal, ENO => #_w1);
   INSERT(EN := #_w1, IN1 := ', ', IN2 := #Name_02, P := 0, OUT => #Column02Internal, ENO => #_w2);
   INSERT(EN := #_w2, IN1 := ', ', IN2 := #Name_03, P := 0, OUT => #Column03Internal, ENO => #_w3);
   INSERT(EN := #_w3, IN1 := ', ', IN2 := #Name_04, P := 0, OUT => #Column04Internal, ENO => #_w4);
   INSERT(EN := #_w4, IN1 := ', ', IN2 := #Name_05, P := 0, OUT => #Column05Internal, ENO => #_w5);
   IF #_w5 THEN INSERT(IN1 := '', IN2 := #Name_06, P := 0, OUT => #Column06Internal); END_IF;
   IF #WriteColumn = 0 THEN
       INSERT(IN1 := #LogColumns, IN2 := #Column01Internal, P := 0, OUT => #LogColumns);
   END_IF;
   IF #WriteColumn = 1 THEN
       INSERT(IN1 := #Column02Internal, IN2 := #LogColumns, P := 0, OUT => #LogColumns);
   END_IF;
   IF #WriteColumn = 2 THEN
       INSERT(IN1 := #Column03Internal, IN2 := #LogColumns, P := 0, OUT => #LogColumns);
   END_IF;
   IF #WriteColumn = 3 THEN
       INSERT(IN1 := #Column04Internal, IN2 := #LogColumns, P := 0, OUT => #LogColumns);
   END_IF;
   IF #WriteColumn = 4 THEN
       INSERT(IN1 := #Column05Internal, IN2 := #LogColumns, P := 0, OUT => #LogColumns);
   END_IF;
   IF #WriteColumn = 5 THEN
       INSERT(IN1 := #Column06Internal, IN2 := #LogColumns, P := 0, OUT => #LogColumns);
   END_IF;
   IF #WriteColumn < 6 THEN #WriteColumn := #WriteColumn + 1; END_IF;
   #WriteColumnReady := #WriteColumn = 6;
END_REGION

REGION Network 4: Data Logging Transfer
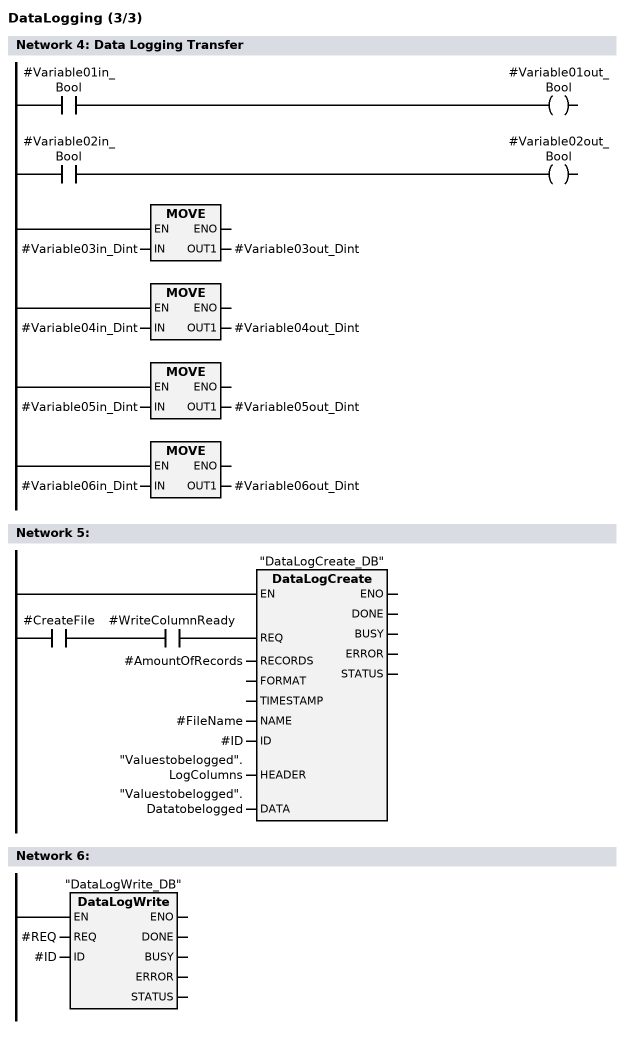
   RUNG wire#powerrail
      Contact( #Variable01in_Bool )
      Coil( #Variable01out_Bool )
   END_RUNG
   RUNG wire#powerrail
      Contact( #Variable02in_Bool )
      Coil( #Variable02out_Bool )
   END_RUNG
   RUNG wire#powerrail
      Move(in := #Variable03in_Dint, out1 => #Variable03out_Dint)
   END_RUNG
   RUNG wire#powerrail
      Move(in := #Variable04in_Dint, out1 => #Variable04out_Dint)
   END_RUNG
   RUNG wire#powerrail
      Move(in := #Variable05in_Dint, out1 => #Variable05out_Dint)
   END_RUNG
   RUNG wire#powerrail
      Move(in := #Variable06in_Dint, out1 => #Variable06out_Dint)
   END_RUNG
   // the same network as SCL:
   #Variable01out_Bool := #Variable01in_Bool;
   #Variable02out_Bool := #Variable02in_Bool;
   #Variable03out_Dint := #Variable03in_Dint;
   #Variable04out_Dint := #Variable04in_Dint;
   #Variable05out_Dint := #Variable05in_Dint;
   #Variable06out_Dint := #Variable06in_Dint;
END_REGION

REGION Network 5
   RUNG wire#powerrail
      "DataLogCreate_DB".DataLogCreate(REQ := wire#w1, RECORDS := #AmountOfRecords, FORMAT :=, TIMESTAMP :=, "NAME" := #FileName, ID := #ID, HEADER := "Valuestobelogged".LogColumns, DATA := "Valuestobelogged".Datatobelogged, DONE =>, BUSY =>, ERROR =>, STATUS =>)
   END_RUNG
   RUNG wire#powerrail
      Contact( #CreateFile )
      Contact( #WriteColumnReady )
   END_RUNG wire#w1
   // the same network as SCL:
   "DataLogCreate_DB"(REQ := #CreateFile AND #WriteColumnReady,   // DataLogCreate
                      RECORDS := #AmountOfRecords,
                      "NAME" := #FileName,
                      ID := #ID,
                      HEADER := "Valuestobelogged".LogColumns,
                      DATA := "Valuestobelogged".Datatobelogged);
END_REGION

REGION Network 6
   RUNG wire#powerrail
      "DataLogWrite_DB".DataLogWrite(REQ := #REQ, ID := #ID, DONE =>, BUSY =>, ERROR =>, STATUS =>)
   END_RUNG
   // the same network as SCL:
   "DataLogWrite_DB"(REQ := #REQ, ID := #ID);   // DataLogWrite
END_REGION
END_FUNCTION_BLOCK

FUNCTION_BLOCK "ZAxis_RelativeMotion_Test"   // FB25, LAD
{ S7_Optimized_Access := 'TRUE' }
VERSION : 0.1
   VAR_INPUT
      StartTest : Bool;
      EndTest : Bool;
      AmountOfSteps : DInt := 3000;
      StepSizeInput : DInt := 100;
      Position : DInt := 0;
      AxisMoving : Bool;
   END_VAR
   VAR_OUTPUT
      StartTask : Bool;
      StepSize : DInt;
      StepNumber : DInt;
      CreateLogFile : Bool;
      StartLog : Bool;
      Comment : String;
   END_VAR
   VAR
      TestActiveInternal : Bool;
      ActualStep : DInt := 9999;
      StepCountNext : DInt := 1;
      MovingInternal : Bool;
      ChangingCount : Bool;
      StartTaskM : Bool;
      LogCreatingReady : Bool;
   END_VAR
BEGIN

REGION Network 1: Log Creating
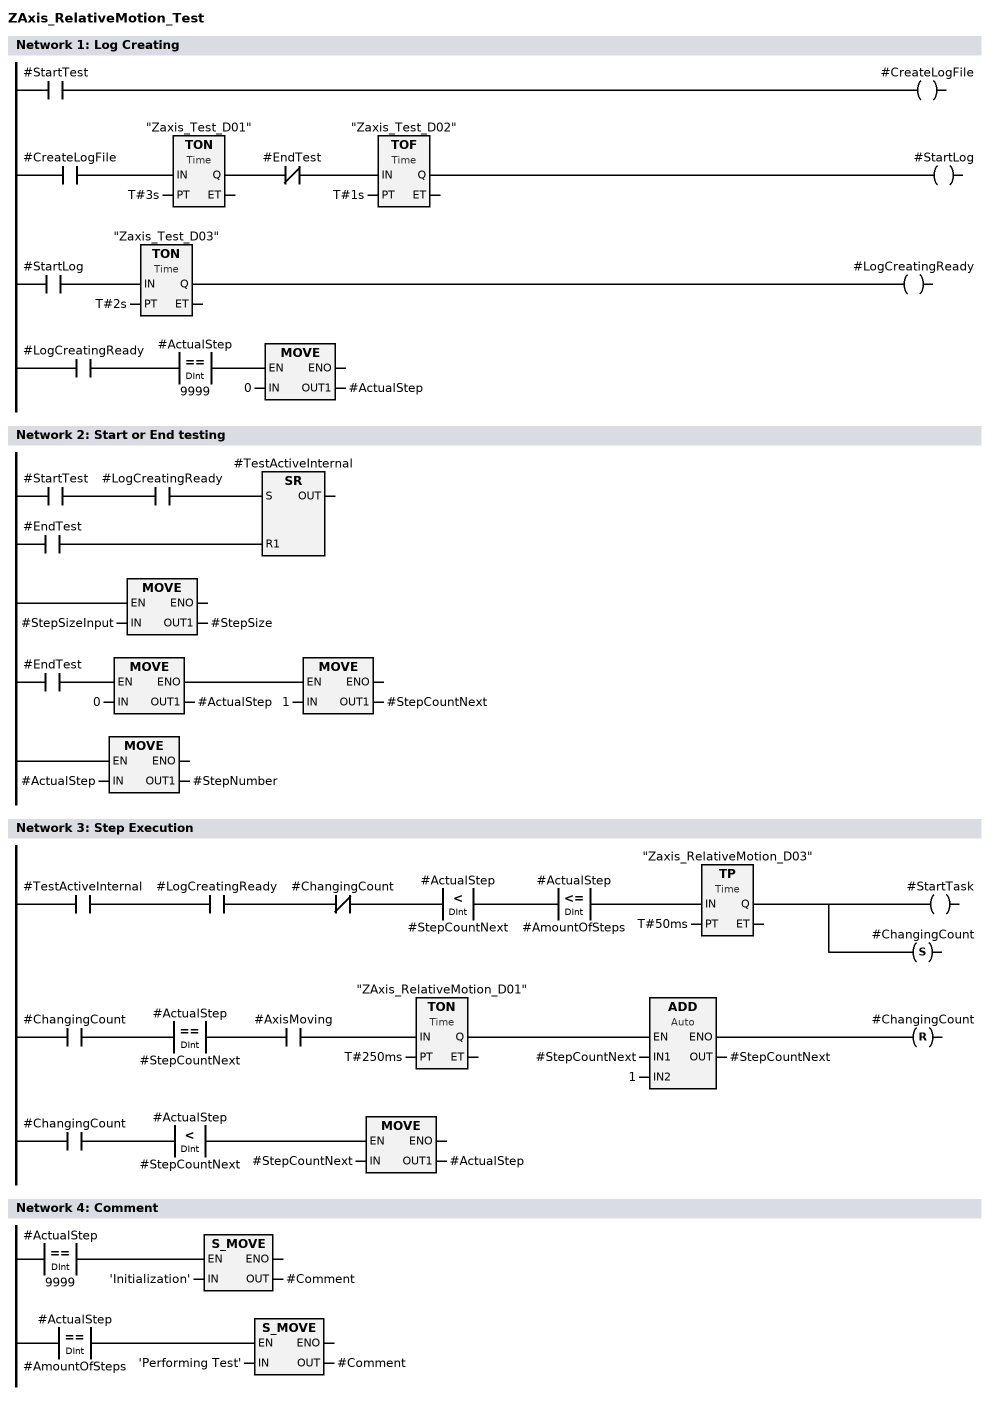
   RUNG wire#powerrail
      Contact( #StartTest )
      Coil( #CreateLogFile )
   END_RUNG
   RUNG wire#powerrail
      Contact( #CreateLogFile )
      { S7_Templates := "time_type := Time" } "Zaxis_Test_D01".TON(pt := T#3s, et =>)
      I_Contact( #EndTest )
      { S7_Templates := "time_type := Time" } "Zaxis_Test_D02".TOF(pt := T#1s, et =>)
      Coil( #StartLog )
   END_RUNG
   RUNG wire#powerrail
      Contact( #StartLog )
      { S7_Templates := "time_type := Time" } "Zaxis_Test_D03".TON(pt := T#2s, et =>)
      Coil( #LogCreatingReady )
   END_RUNG
   RUNG wire#powerrail
      Contact( #LogCreatingReady )
      { S7_Templates := "SrcType := DInt" } EQ_Contact(in1 := #ActualStep, in2 := 9999)
      Move(in := 0, out1 => #ActualStep)
   END_RUNG
   // the same network as SCL:
   #CreateLogFile := #StartTest;
   "Zaxis_Test_D01".TON(IN := #CreateLogFile, PT := T#3s);
   "Zaxis_Test_D02".TOF(IN := "Zaxis_Test_D01".Q AND NOT #EndTest, PT := T#1s);
   #StartLog := "Zaxis_Test_D02".Q;
   "Zaxis_Test_D03".TON(IN := #StartLog, PT := T#2s);
   #LogCreatingReady := "Zaxis_Test_D03".Q;
   IF #LogCreatingReady AND (#ActualStep = 9999) THEN #ActualStep := 0; END_IF;
END_REGION

REGION Network 2: Start or End testing
   RUNG wire#powerrail
      Contact( #StartTest )
      Contact( #LogCreatingReady )
      S_SR(operand := #TestActiveInternal, r1 := wire#w1)
   END_RUNG
   RUNG wire#powerrail
      Contact( #EndTest )
   END_RUNG wire#w1
   RUNG wire#powerrail
      Move(in := #StepSizeInput, out1 => #StepSize)
   END_RUNG
   RUNG wire#powerrail
      Contact( #EndTest )
      Move(in := 0, out1 => #ActualStep)
      Move(in := 1, out1 => #StepCountNext)
   END_RUNG
   RUNG wire#powerrail
      Move(in := #ActualStep, out1 => #StepNumber)
   END_RUNG
   // the same network as SCL:
   IF #StartTest AND #LogCreatingReady THEN
       #TestActiveInternal := TRUE;   // SR flip-flop
   END_IF;
   IF #EndTest THEN #TestActiveInternal := FALSE; END_IF;
   #StepSize := #StepSizeInput;
   IF #EndTest THEN
       #ActualStep := 0;
       #StepCountNext := 1;
   END_IF;
   #StepNumber := #ActualStep;
END_REGION

REGION Network 3: Step Execution
   RUNG wire#powerrail
      Contact( #TestActiveInternal )
      Contact( #LogCreatingReady )
      I_Contact( #ChangingCount )
      { S7_Templates := "SrcType := DInt" } LT_Contact(in1 := #ActualStep, in2 := #StepCountNext)
      { S7_Templates := "SrcType := DInt" } LE_Contact(in1 := #ActualStep, in2 := #AmountOfSteps)
      { S7_Templates := "time_type := Time" } "Zaxis_RelativeMotion_D03".TP(pt := T#50ms, et =>)
      wire#w1
      Coil( #StartTask )
   END_RUNG
   RUNG wire#w1
      S_Coil( #ChangingCount )
   END_RUNG
   RUNG wire#powerrail
      Contact( #ChangingCount )
      { S7_Templates := "SrcType := DInt" } EQ_Contact(in1 := #ActualStep, in2 := #StepCountNext)
      Contact( #AxisMoving )
      { S7_Templates := "time_type := Time" } "ZAxis_RelativeMotion_D01".TON(pt := T#250ms, et =>)
      Add(in1 := #StepCountNext, in2 := 1, out => #StepCountNext)
      R_Coil( #ChangingCount )
   END_RUNG
   RUNG wire#powerrail
      Contact( #ChangingCount )
      { S7_Templates := "SrcType := DInt" } LT_Contact(in1 := #ActualStep, in2 := #StepCountNext)
      Move(in := #StepCountNext, out1 => #ActualStep)
   END_RUNG
   // the same network as SCL:
   "Zaxis_RelativeMotion_D03".TP(IN := #TestActiveInternal AND #LogCreatingReady AND NOT #ChangingCount AND (#ActualStep < #StepCountNext) AND (#ActualStep <= #AmountOfSteps),
                           PT := T#50ms);
   #StartTask := "Zaxis_RelativeMotion_D03".Q;
   IF "Zaxis_RelativeMotion_D03".Q THEN #ChangingCount := TRUE; END_IF;
   "ZAxis_RelativeMotion_D01".TON(IN := #ChangingCount AND (#ActualStep = #StepCountNext) AND #AxisMoving,
                           PT := T#250ms);
   IF "ZAxis_RelativeMotion_D01".Q THEN
       #StepCountNext := #StepCountNext + 1;
       #ChangingCount := FALSE;
   END_IF;
   IF #ChangingCount AND (#ActualStep < #StepCountNext) THEN #ActualStep := #StepCountNext; END_IF;
END_REGION

REGION Network 4: Comment
   RUNG wire#powerrail
      { S7_Templates := "SrcType := DInt" } EQ_Contact(in1 := #ActualStep, in2 := 9999)
      S_Move(in := 'Initialization', out => #Comment)
   END_RUNG
   RUNG wire#powerrail
      { S7_Templates := "SrcType := DInt" } EQ_Contact(in1 := #ActualStep, in2 := #AmountOfSteps)
      S_Move(in := 'Performing Test', out => #Comment)
   END_RUNG
   // the same network as SCL:
   IF #ActualStep = 9999 THEN #Comment := 'Initialization'; END_IF;
   IF #ActualStep = #AmountOfSteps THEN #Comment := 'Performing Test'; END_IF;
END_REGION
END_FUNCTION_BLOCK

ORGANIZATION_BLOCK "Work Cyclic"   // OB30, LAD, CyclicInterrupt
TITLE = Description:
{ S7_Optimized_Access := 'TRUE' }
VERSION : 0.1
// Operations that are supposed to be executed in a precise cycle time, which is temporary set to 45ms. It is important to connect this time with the read/write time of the WebDB (NOAH).
   VAR_INPUT
      Initial_Call : Bool;   // Initial call of this OB
      Event_Count : Int;   // Events discarded
   END_VAR
   VAR_TEMP   // added for the SCL form of the ladder/FBD networks
      _w1 : Bool;
   END_VAR
BEGIN

REGION Network 1: AXIS Z1 Control CMMT V2 To Update
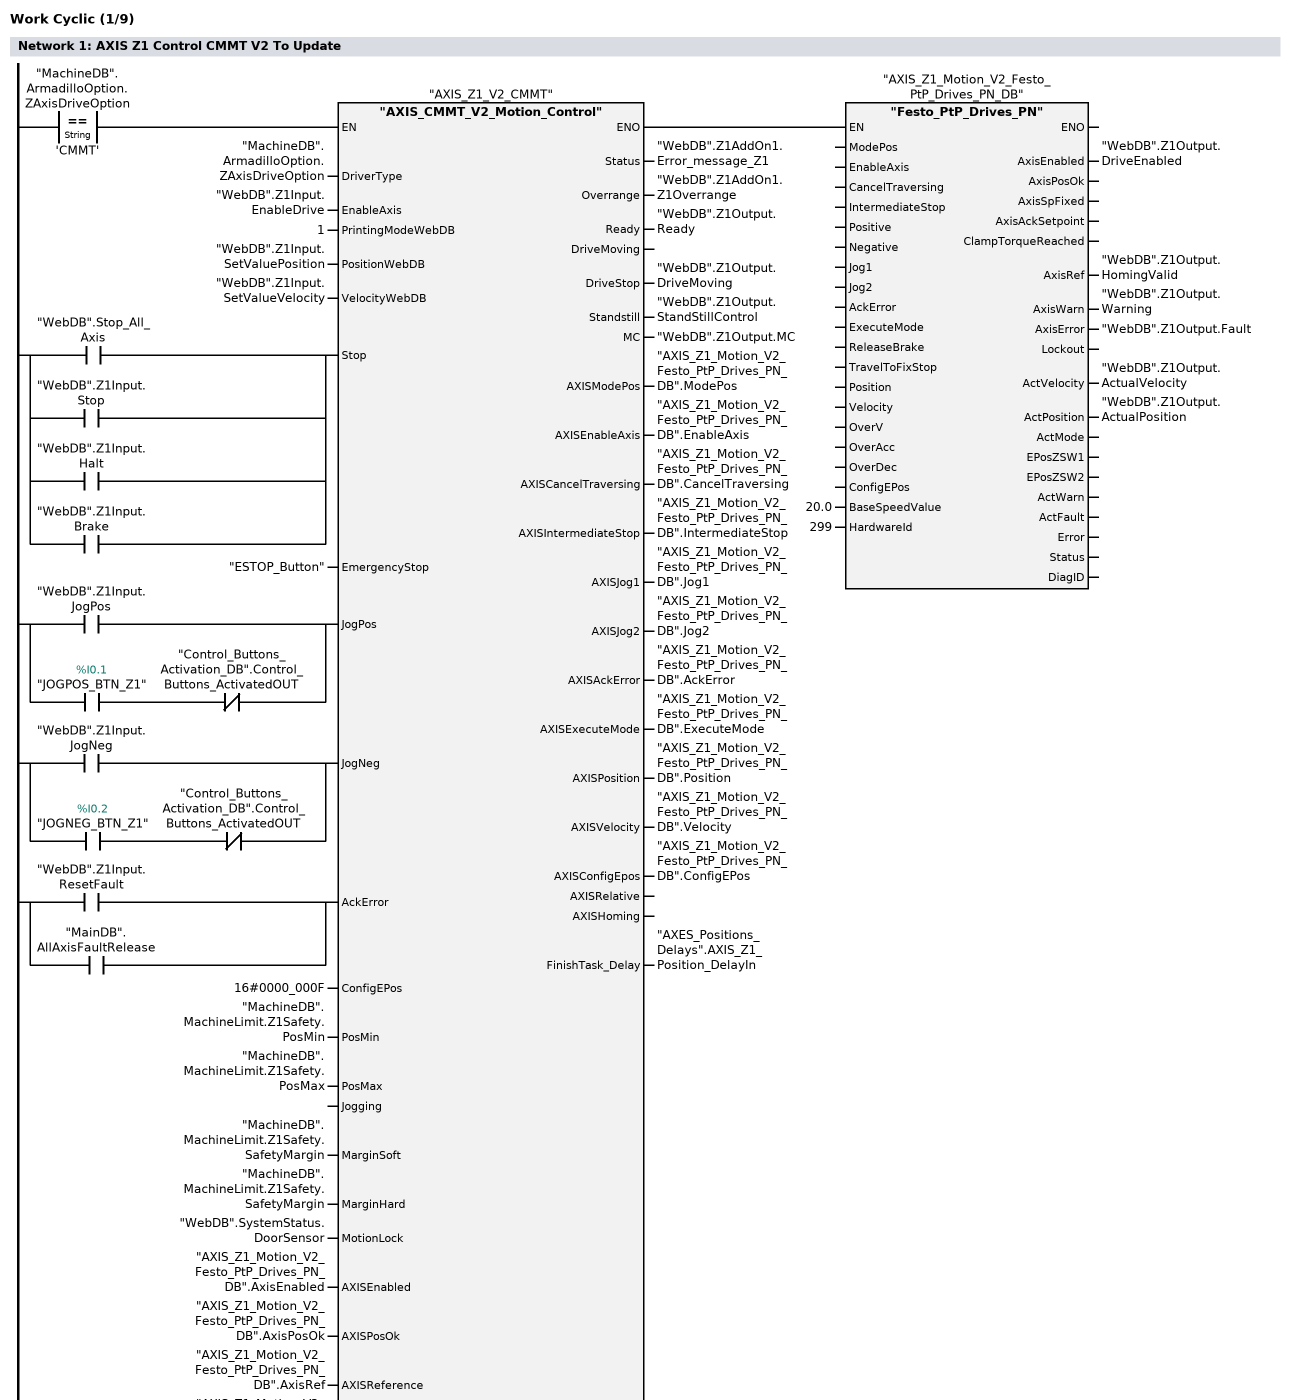
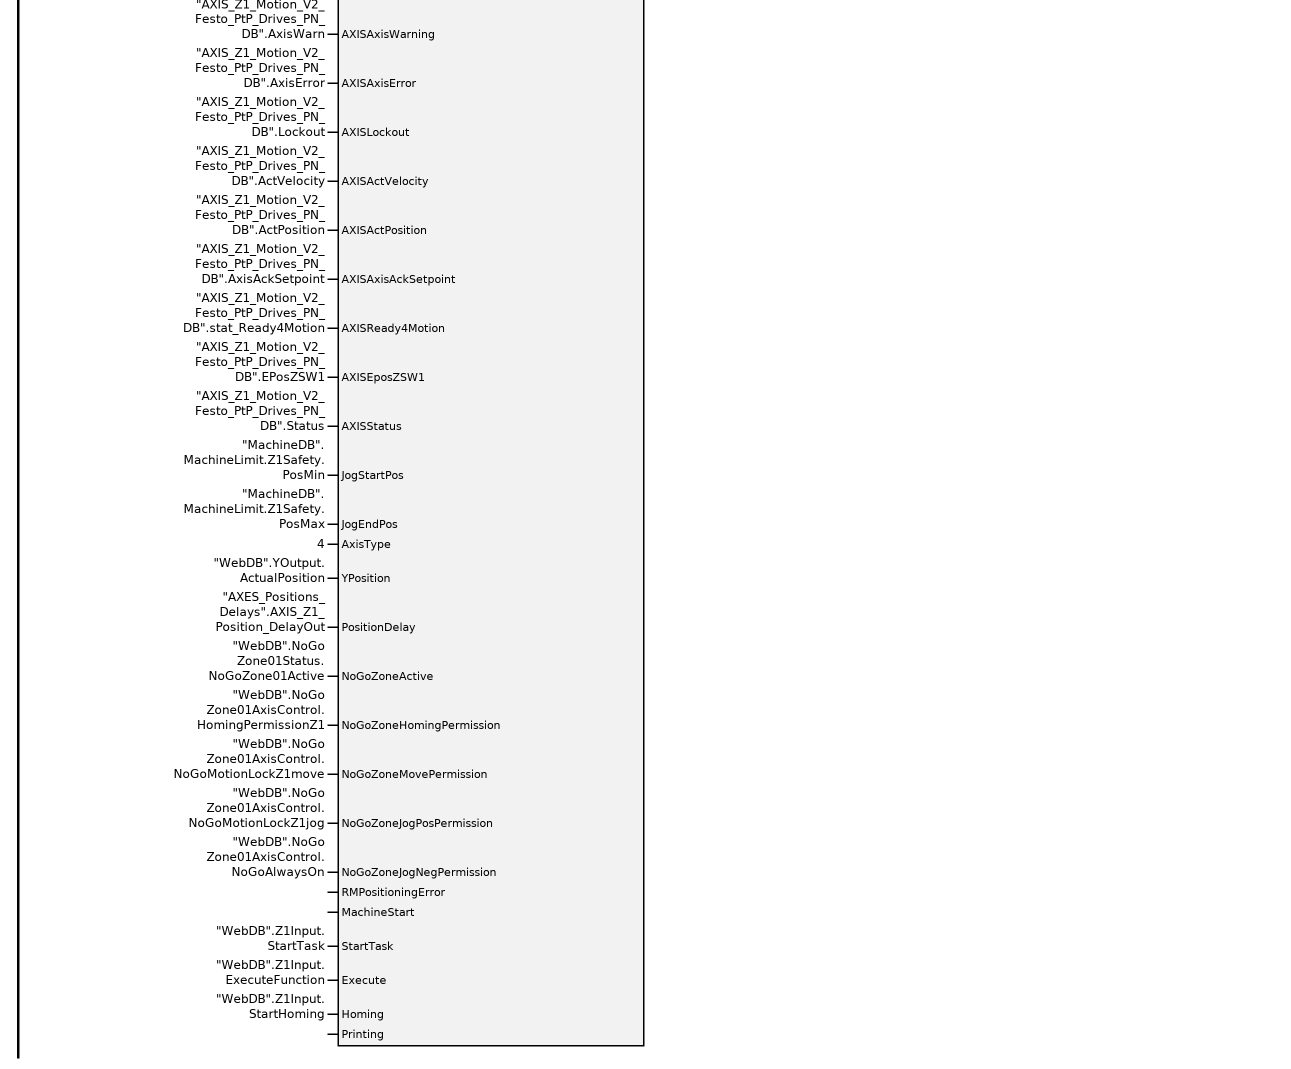
   RUNG wire#powerrail
      { S7_Templates := "SrcType := String" } EQ_Contact(in1 := "MachineDB".ArmadilloOption.ZAxisDriveOption, in2 := 'CMMT')
      "AXIS_Z1_V2_CMMT"(Stop := wire#w1, JogPos := wire#w2, JogNeg := wire#w3, AckError := wire#w4, DriverType := "MachineDB".ArmadilloOption.ZAxisDriveOption, EnableAxis := "WebDB".Z1Input.EnableDrive, PrintingModeWebDB := 1, PositionWebDB := "WebDB".Z1Input.SetValuePosition, VelocityWebDB := "WebDB".Z1Input.SetValueVelocity, EmergencyStop := "ESTOP_Button", ConfigEPos := 16#0000_000F, PosMin := "MachineDB".MachineLimit.Z1Safety.PosMin, PosMax := "MachineDB".MachineLimit.Z1Safety.PosMax, Jogging :=, MarginSoft := "MachineDB".MachineLimit.Z1Safety.SafetyMargin, MarginHard := "MachineDB".MachineLimit.Z1Safety.SafetyMargin, MotionLock := "WebDB".SystemStatus.DoorSensor, AXISEnabled := "AXIS_Z1_Motion_V2_Festo_PtP_Drives_PN_DB".AxisEnabled, AXISPosOk := "AXIS_Z1_Motion_V2_Festo_PtP_Drives_PN_DB".AxisPosOk, AXISReference := "AXIS_Z1_Motion_V2_Festo_PtP_Drives_PN_DB".AxisRef, AXISAxisWarning := "AXIS_Z1_Motion_V2_Festo_PtP_Drives_PN_DB".AxisWarn, AXISAxisError := "AXIS_Z1_Motion_V2_Festo_PtP_Drives_PN_DB".AxisError, AXISLockout := "AXIS_Z1_Motion_V2_Festo_PtP_Drives_PN_DB".Lockout, AXISActVelocity := "AXIS_Z1_Motion_V2_Festo_PtP_Drives_PN_DB".ActVelocity, AXISActPosition := "AXIS_Z1_Motion_V2_Festo_PtP_Drives_PN_DB".ActPosition, AXISAxisAckSetpoint := "AXIS_Z1_Motion_V2_Festo_PtP_Drives_PN_DB".AxisAckSetpoint, AXISReady4Motion := "AXIS_Z1_Motion_V2_Festo_PtP_Drives_PN_DB".stat_Ready4Motion, AXISEposZSW1 := "AXIS_Z1_Motion_V2_Festo_PtP_Drives_PN_DB".EPosZSW1, AXISStatus := "AXIS_Z1_Motion_V2_Festo_PtP_Drives_PN_DB".Status, JogStartPos := "MachineDB".MachineLimit.Z1Safety.PosMin, JogEndPos := "MachineDB".MachineLimit.Z1Safety.PosMax, AxisType := 4, YPosition := "WebDB".YOutput.ActualPosition, PositionDelay := "AXES_Positions_Delays".AXIS_Z1_Position_DelayOut, NoGoZoneActive := "WebDB".NoGoZone01Status.NoGoZone01Active, NoGoZoneHomingPermission := "WebDB".NoGoZone01AxisControl.HomingPermissionZ1, NoGoZoneMovePermission := "WebDB".NoGoZone01AxisControl.NoGoMotionLockZ1move, NoGoZoneJogPosPermission := "WebDB".NoGoZone01AxisControl.NoGoMotionLockZ1jog, NoGoZoneJogNegPermission := "WebDB".NoGoZone01AxisControl.NoGoAlwaysOn, RMPositioningError :=, MachineStart :=, StartTask := "WebDB".Z1Input.StartTask, Execute := "WebDB".Z1Input.ExecuteFunction, Homing := "WebDB".Z1Input.StartHoming, Printing :=, Status => "WebDB".Z1AddOn1.Error_message_Z1, Overrange => "WebDB".Z1AddOn1.Z1Overrange, Ready => "WebDB".Z1Output.Ready, DriveMoving =>, DriveStop => "WebDB".Z1Output.DriveMoving, Standstill => "WebDB".Z1Output.StandStillControl, MC => "WebDB".Z1Output.MC, AXISModePos => "AXIS_Z1_Motion_V2_Festo_PtP_Drives_PN_DB".ModePos, AXISEnableAxis => "AXIS_Z1_Motion_V2_Festo_PtP_Drives_PN_DB".EnableAxis, AXISCancelTraversing => "AXIS_Z1_Motion_V2_Festo_PtP_Drives_PN_DB".CancelTraversing, AXISIntermediateStop => "AXIS_Z1_Motion_V2_Festo_PtP_Drives_PN_DB".IntermediateStop, AXISJog1 => "AXIS_Z1_Motion_V2_Festo_PtP_Drives_PN_DB".Jog1, AXISJog2 => "AXIS_Z1_Motion_V2_Festo_PtP_Drives_PN_DB".Jog2, AXISAckError => "AXIS_Z1_Motion_V2_Festo_PtP_Drives_PN_DB".AckError, AXISExecuteMode => "AXIS_Z1_Motion_V2_Festo_PtP_Drives_PN_DB".ExecuteMode, AXISPosition => "AXIS_Z1_Motion_V2_Festo_PtP_Drives_PN_DB".Position, AXISVelocity => "AXIS_Z1_Motion_V2_Festo_PtP_Drives_PN_DB".Velocity, AXISConfigEpos => "AXIS_Z1_Motion_V2_Festo_PtP_Drives_PN_DB".ConfigEPos, AXISRelative =>, AXISHoming =>, FinishTask_Delay => "AXES_Positions_Delays".AXIS_Z1_Position_DelayIn)
      "AXIS_Z1_Motion_V2_Festo_PtP_Drives_PN_DB"(ModePos :=, EnableAxis :=, CancelTraversing :=, IntermediateStop :=, Positive :=, Negative :=, Jog1 :=, Jog2 :=, AckError :=, ExecuteMode :=, ReleaseBrake :=, TravelToFixStop :=, Position :=, Velocity :=, OverV :=, OverAcc :=, OverDec :=, ConfigEPos :=, BaseSpeedValue := 20.0, HardwareId := 299, AxisEnabled => "WebDB".Z1Output.DriveEnabled, AxisPosOk =>, AxisSpFixed =>, AxisAckSetpoint =>, ClampTorqueReached =>, AxisRef => "WebDB".Z1Output.HomingValid, AxisWarn => "WebDB".Z1Output.Warning, AxisError => "WebDB".Z1Output.Fault, Lockout =>, ActVelocity => "WebDB".Z1Output.ActualVelocity, ActPosition => "WebDB".Z1Output.ActualPosition, ActMode =>, EPosZSW1 =>, EPosZSW2 =>, ActWarn =>, ActFault =>, Error =>, Status =>, DiagID =>)
   END_RUNG
   RUNG wire#powerrail
      Contact( "WebDB".Stop_All_Axis )
   END_RUNG wire#w1
   RUNG wire#powerrail
      Contact( "WebDB".Z1Input.Stop )
   END_RUNG wire#w1
   RUNG wire#powerrail
      Contact( "WebDB".Z1Input.Halt )
   END_RUNG wire#w1
   RUNG wire#powerrail
      Contact( "WebDB".Z1Input.Brake )
   END_RUNG wire#w1
   RUNG wire#powerrail
      Contact( "WebDB".Z1Input.JogPos )
   END_RUNG wire#w2
   RUNG wire#powerrail
      Contact( "JOGPOS_BTN_Z1" )
      I_Contact( "Control_Buttons_Activation_DB".Control_Buttons_ActivatedOUT )
   END_RUNG wire#w2
   RUNG wire#powerrail
      Contact( "WebDB".Z1Input.JogNeg )
   END_RUNG wire#w3
   RUNG wire#powerrail
      Contact( "JOGNEG_BTN_Z1" )
      I_Contact( "Control_Buttons_Activation_DB".Control_Buttons_ActivatedOUT )
   END_RUNG wire#w3
   RUNG wire#powerrail
      Contact( "WebDB".Z1Input.ResetFault )
   END_RUNG wire#w4
   RUNG wire#powerrail
      Contact( "MainDB".AllAxisFaultRelease )
   END_RUNG wire#w4
   // the same network as SCL:
   "AXIS_Z1_V2_CMMT"(EN := "MachineDB".ArmadilloOption.ZAxisDriveOption = 'CMMT',   // "AXIS_CMMT_V2_Motion_Control"
                     DriverType := "MachineDB".ArmadilloOption.ZAxisDriveOption,
                     EnableAxis := "WebDB".Z1Input.EnableDrive,
                     PrintingModeWebDB := 1,
                     PositionWebDB := "WebDB".Z1Input.SetValuePosition,
                     VelocityWebDB := "WebDB".Z1Input.SetValueVelocity,
                     Stop := "WebDB".Stop_All_Axis OR "WebDB".Z1Input.Stop OR "WebDB".Z1Input.Halt OR "WebDB".Z1Input.Brake,
                     EmergencyStop := "ESTOP_Button",
                     JogPos := "WebDB".Z1Input.JogPos OR ("JOGPOS_BTN_Z1" AND NOT "Control_Buttons_Activation_DB".Control_Buttons_ActivatedOUT),
                     JogNeg := "WebDB".Z1Input.JogNeg OR ("JOGNEG_BTN_Z1" AND NOT "Control_Buttons_Activation_DB".Control_Buttons_ActivatedOUT),
                     AckError := "WebDB".Z1Input.ResetFault OR "MainDB".AllAxisFaultRelease,
                     ConfigEPos := 16#0000_000F,
                     PosMin := "MachineDB".MachineLimit.Z1Safety.PosMin,
                     PosMax := "MachineDB".MachineLimit.Z1Safety.PosMax,
                     MarginSoft := "MachineDB".MachineLimit.Z1Safety.SafetyMargin,
                     MarginHard := "MachineDB".MachineLimit.Z1Safety.SafetyMargin,
                     MotionLock := "WebDB".SystemStatus.DoorSensor,
                     AXISEnabled := "AXIS_Z1_Motion_V2_Festo_PtP_Drives_PN_DB".AxisEnabled,
                     AXISPosOk := "AXIS_Z1_Motion_V2_Festo_PtP_Drives_PN_DB".AxisPosOk,
                     AXISReference := "AXIS_Z1_Motion_V2_Festo_PtP_Drives_PN_DB".AxisRef,
                     AXISAxisWarning := "AXIS_Z1_Motion_V2_Festo_PtP_Drives_PN_DB".AxisWarn,
                     AXISAxisError := "AXIS_Z1_Motion_V2_Festo_PtP_Drives_PN_DB".AxisError,
                     AXISLockout := "AXIS_Z1_Motion_V2_Festo_PtP_Drives_PN_DB".Lockout,
                     AXISActVelocity := "AXIS_Z1_Motion_V2_Festo_PtP_Drives_PN_DB".ActVelocity,
                     AXISActPosition := "AXIS_Z1_Motion_V2_Festo_PtP_Drives_PN_DB".ActPosition,
                     AXISAxisAckSetpoint := "AXIS_Z1_Motion_V2_Festo_PtP_Drives_PN_DB".AxisAckSetpoint,
                     AXISReady4Motion := "AXIS_Z1_Motion_V2_Festo_PtP_Drives_PN_DB".stat_Ready4Motion,
                     AXISEposZSW1 := "AXIS_Z1_Motion_V2_Festo_PtP_Drives_PN_DB".EPosZSW1,
                     AXISStatus := "AXIS_Z1_Motion_V2_Festo_PtP_Drives_PN_DB".Status,
                     JogStartPos := "MachineDB".MachineLimit.Z1Safety.PosMin,
                     JogEndPos := "MachineDB".MachineLimit.Z1Safety.PosMax,
                     AxisType := 4,
                     YPosition := "WebDB".YOutput.ActualPosition,
                     PositionDelay := "AXES_Positions_Delays".AXIS_Z1_Position_DelayOut,
                     NoGoZoneActive := "WebDB".NoGoZone01Status.NoGoZone01Active,
                     NoGoZoneHomingPermission := "WebDB".NoGoZone01AxisControl.HomingPermissionZ1,
                     NoGoZoneMovePermission := "WebDB".NoGoZone01AxisControl.NoGoMotionLockZ1move,
                     NoGoZoneJogPosPermission := "WebDB".NoGoZone01AxisControl.NoGoMotionLockZ1jog,
                     NoGoZoneJogNegPermission := "WebDB".NoGoZone01AxisControl.NoGoAlwaysOn,
                     StartTask := "WebDB".Z1Input.StartTask,
                     Execute := "WebDB".Z1Input.ExecuteFunction,
                     Homing := "WebDB".Z1Input.StartHoming,
                     Status => "WebDB".Z1AddOn1.Error_message_Z1,
                     Overrange => "WebDB".Z1AddOn1.Z1Overrange,
                     Ready => "WebDB".Z1Output.Ready,
                     DriveStop => "WebDB".Z1Output.DriveMoving,
                     Standstill => "WebDB".Z1Output.StandStillControl,
                     MC => "WebDB".Z1Output.MC,
                     AXISModePos => "AXIS_Z1_Motion_V2_Festo_PtP_Drives_PN_DB".ModePos,
                     AXISEnableAxis => "AXIS_Z1_Motion_V2_Festo_PtP_Drives_PN_DB".EnableAxis,
                     AXISCancelTraversing => "AXIS_Z1_Motion_V2_Festo_PtP_Drives_PN_DB".CancelTraversing,
                     AXISIntermediateStop => "AXIS_Z1_Motion_V2_Festo_PtP_Drives_PN_DB".IntermediateStop,
                     AXISJog1 => "AXIS_Z1_Motion_V2_Festo_PtP_Drives_PN_DB".Jog1,
                     AXISJog2 => "AXIS_Z1_Motion_V2_Festo_PtP_Drives_PN_DB".Jog2,
                     AXISAckError => "AXIS_Z1_Motion_V2_Festo_PtP_Drives_PN_DB".AckError,
                     AXISExecuteMode => "AXIS_Z1_Motion_V2_Festo_PtP_Drives_PN_DB".ExecuteMode,
                     AXISPosition => "AXIS_Z1_Motion_V2_Festo_PtP_Drives_PN_DB".Position,
                     AXISVelocity => "AXIS_Z1_Motion_V2_Festo_PtP_Drives_PN_DB".Velocity,
                     AXISConfigEpos => "AXIS_Z1_Motion_V2_Festo_PtP_Drives_PN_DB".ConfigEPos,
                     FinishTask_Delay => "AXES_Positions_Delays".AXIS_Z1_Position_DelayIn,
                     ENO => #_w1);
   IF #_w1 THEN
       "AXIS_Z1_Motion_V2_Festo_PtP_Drives_PN_DB"(BaseSpeedValue := 20.0,   // "Festo_PtP_Drives_PN"
                               HardwareId := 299,
                               AxisEnabled => "WebDB".Z1Output.DriveEnabled,
                               AxisRef => "WebDB".Z1Output.HomingValid,
                               AxisWarn => "WebDB".Z1Output.Warning,
                               AxisError => "WebDB".Z1Output.Fault,
                               ActVelocity => "WebDB".Z1Output.ActualVelocity,
                               ActPosition => "WebDB".Z1Output.ActualPosition);
   END_IF;
END_REGION

REGION Network 2: AXIS Z1 Control CMMS
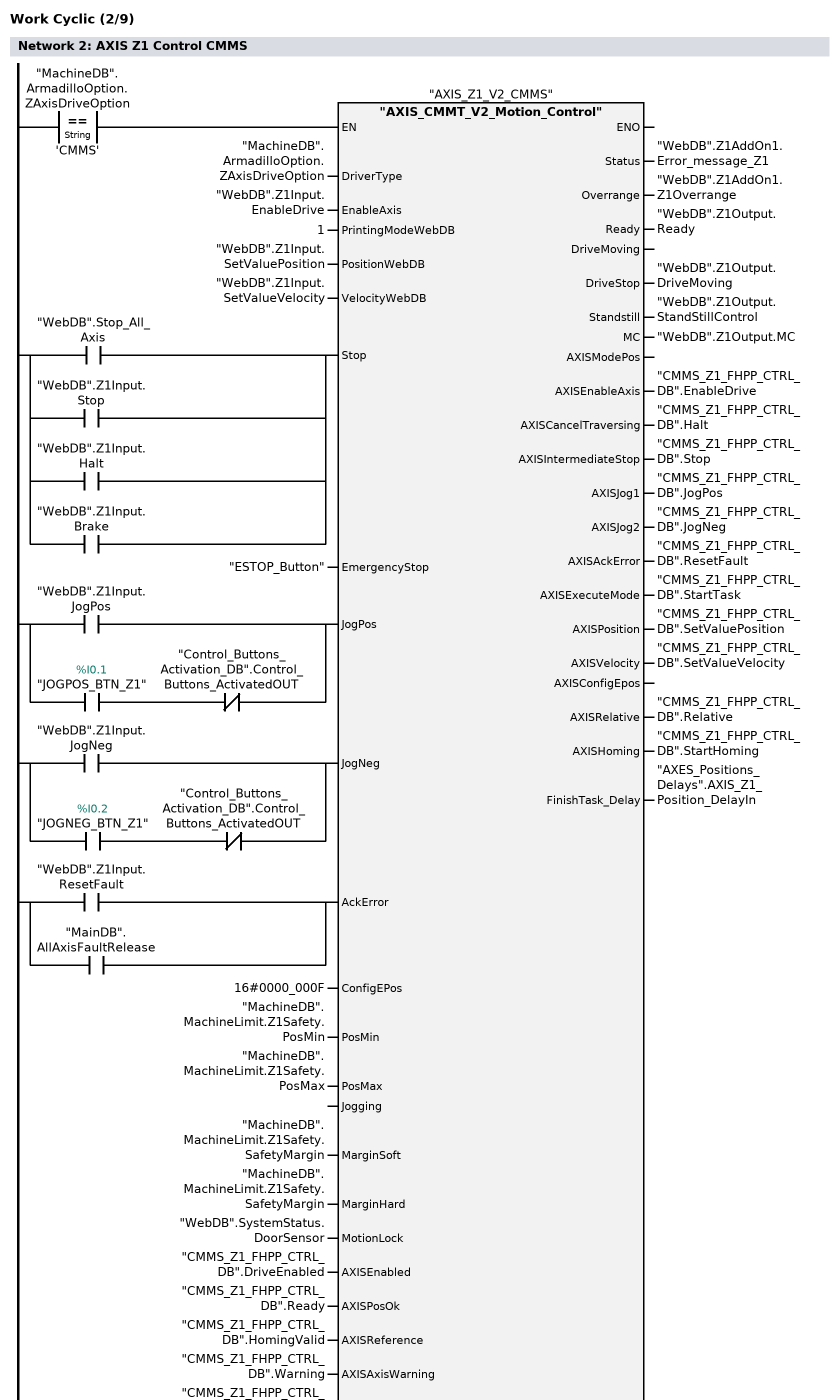
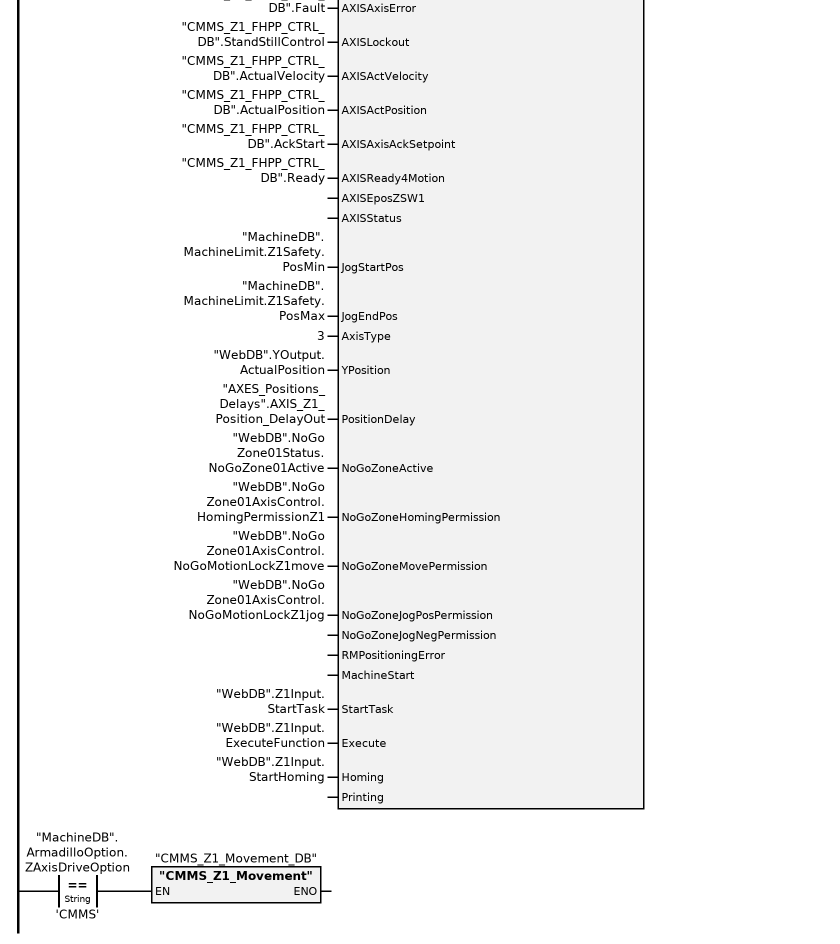
   RUNG wire#powerrail
      { S7_Templates := "SrcType := String" } EQ_Contact(in1 := "MachineDB".ArmadilloOption.ZAxisDriveOption, in2 := 'CMMS')
      "AXIS_Z1_V2_CMMS"(Stop := wire#w1, JogPos := wire#w2, JogNeg := wire#w3, AckError := wire#w4, DriverType := "MachineDB".ArmadilloOption.ZAxisDriveOption, EnableAxis := "WebDB".Z1Input.EnableDrive, PrintingModeWebDB := 1, PositionWebDB := "WebDB".Z1Input.SetValuePosition, VelocityWebDB := "WebDB".Z1Input.SetValueVelocity, EmergencyStop := "ESTOP_Button", ConfigEPos := 16#0000_000F, PosMin := "MachineDB".MachineLimit.Z1Safety.PosMin, PosMax := "MachineDB".MachineLimit.Z1Safety.PosMax, Jogging :=, MarginSoft := "MachineDB".MachineLimit.Z1Safety.SafetyMargin, MarginHard := "MachineDB".MachineLimit.Z1Safety.SafetyMargin, MotionLock := "WebDB".SystemStatus.DoorSensor, AXISEnabled := "CMMS_Z1_FHPP_CTRL_DB".DriveEnabled, AXISPosOk := "CMMS_Z1_FHPP_CTRL_DB".Ready, AXISReference := "CMMS_Z1_FHPP_CTRL_DB".HomingValid, AXISAxisWarning := "CMMS_Z1_FHPP_CTRL_DB".Warning, AXISAxisError := "CMMS_Z1_FHPP_CTRL_DB".Fault, AXISLockout := "CMMS_Z1_FHPP_CTRL_DB".StandStillControl, AXISActVelocity := "CMMS_Z1_FHPP_CTRL_DB".ActualVelocity, AXISActPosition := "CMMS_Z1_FHPP_CTRL_DB".ActualPosition, AXISAxisAckSetpoint := "CMMS_Z1_FHPP_CTRL_DB".AckStart, AXISReady4Motion := "CMMS_Z1_FHPP_CTRL_DB".Ready, AXISEposZSW1 :=, AXISStatus :=, JogStartPos := "MachineDB".MachineLimit.Z1Safety.PosMin, JogEndPos := "MachineDB".MachineLimit.Z1Safety.PosMax, AxisType := 3, YPosition := "WebDB".YOutput.ActualPosition, PositionDelay := "AXES_Positions_Delays".AXIS_Z1_Position_DelayOut, NoGoZoneActive := "WebDB".NoGoZone01Status.NoGoZone01Active, NoGoZoneHomingPermission := "WebDB".NoGoZone01AxisControl.HomingPermissionZ1, NoGoZoneMovePermission := "WebDB".NoGoZone01AxisControl.NoGoMotionLockZ1move, NoGoZoneJogPosPermission := "WebDB".NoGoZone01AxisControl.NoGoMotionLockZ1jog, NoGoZoneJogNegPermission :=, RMPositioningError :=, MachineStart :=, StartTask := "WebDB".Z1Input.StartTask, Execute := "WebDB".Z1Input.ExecuteFunction, Homing := "WebDB".Z1Input.StartHoming, Printing :=, Status => "WebDB".Z1AddOn1.Error_message_Z1, Overrange => "WebDB".Z1AddOn1.Z1Overrange, Ready => "WebDB".Z1Output.Ready, DriveMoving =>, DriveStop => "WebDB".Z1Output.DriveMoving, Standstill => "WebDB".Z1Output.StandStillControl, MC => "WebDB".Z1Output.MC, AXISModePos =>, AXISEnableAxis => "CMMS_Z1_FHPP_CTRL_DB".EnableDrive, AXISCancelTraversing => "CMMS_Z1_FHPP_CTRL_DB".Halt, AXISIntermediateStop => "CMMS_Z1_FHPP_CTRL_DB".Stop, AXISJog1 => "CMMS_Z1_FHPP_CTRL_DB".JogPos, AXISJog2 => "CMMS_Z1_FHPP_CTRL_DB".JogNeg, AXISAckError => "CMMS_Z1_FHPP_CTRL_DB".ResetFault, AXISExecuteMode => "CMMS_Z1_FHPP_CTRL_DB".StartTask, AXISPosition => "CMMS_Z1_FHPP_CTRL_DB".SetValuePosition, AXISVelocity => "CMMS_Z1_FHPP_CTRL_DB".SetValueVelocity, AXISConfigEpos =>, AXISRelative => "CMMS_Z1_FHPP_CTRL_DB".Relative, AXISHoming => "CMMS_Z1_FHPP_CTRL_DB".StartHoming, FinishTask_Delay => "AXES_Positions_Delays".AXIS_Z1_Position_DelayIn)
   END_RUNG
   RUNG wire#powerrail
      Contact( "WebDB".Stop_All_Axis )
   END_RUNG wire#w1
   RUNG wire#powerrail
      Contact( "WebDB".Z1Input.Stop )
   END_RUNG wire#w1
   RUNG wire#powerrail
      Contact( "WebDB".Z1Input.Halt )
   END_RUNG wire#w1
   RUNG wire#powerrail
      Contact( "WebDB".Z1Input.Brake )
   END_RUNG wire#w1
   RUNG wire#powerrail
      Contact( "WebDB".Z1Input.JogPos )
   END_RUNG wire#w2
   RUNG wire#powerrail
      Contact( "JOGPOS_BTN_Z1" )
      I_Contact( "Control_Buttons_Activation_DB".Control_Buttons_ActivatedOUT )
   END_RUNG wire#w2
   RUNG wire#powerrail
      Contact( "WebDB".Z1Input.JogNeg )
   END_RUNG wire#w3
   RUNG wire#powerrail
      Contact( "JOGNEG_BTN_Z1" )
      I_Contact( "Control_Buttons_Activation_DB".Control_Buttons_ActivatedOUT )
   END_RUNG wire#w3
   RUNG wire#powerrail
      Contact( "WebDB".Z1Input.ResetFault )
   END_RUNG wire#w4
   RUNG wire#powerrail
      Contact( "MainDB".AllAxisFaultRelease )
   END_RUNG wire#w4
   RUNG wire#powerrail
      { S7_Templates := "SrcType := String" } EQ_Contact(in1 := "MachineDB".ArmadilloOption.ZAxisDriveOption, in2 := 'CMMS')
      "CMMS_Z1_Movement_DB"()
   END_RUNG
   // the same network as SCL:
   IF "MachineDB".ArmadilloOption.ZAxisDriveOption = 'CMMS' THEN
       "AXIS_Z1_V2_CMMS"(DriverType := "MachineDB".ArmadilloOption.ZAxisDriveOption,   // "AXIS_CMMT_V2_Motion_Control"
                         EnableAxis := "WebDB".Z1Input.EnableDrive,
                         PrintingModeWebDB := 1,
                         PositionWebDB := "WebDB".Z1Input.SetValuePosition,
                         VelocityWebDB := "WebDB".Z1Input.SetValueVelocity,
                         Stop := "WebDB".Stop_All_Axis OR "WebDB".Z1Input.Stop OR "WebDB".Z1Input.Halt OR "WebDB".Z1Input.Brake,
                         EmergencyStop := "ESTOP_Button",
                         JogPos := "WebDB".Z1Input.JogPos OR ("JOGPOS_BTN_Z1" AND NOT "Control_Buttons_Activation_DB".Control_Buttons_ActivatedOUT),
                         JogNeg := "WebDB".Z1Input.JogNeg OR ("JOGNEG_BTN_Z1" AND NOT "Control_Buttons_Activation_DB".Control_Buttons_ActivatedOUT),
                         AckError := "WebDB".Z1Input.ResetFault OR "MainDB".AllAxisFaultRelease,
                         ConfigEPos := 16#0000_000F,
                         PosMin := "MachineDB".MachineLimit.Z1Safety.PosMin,
                         PosMax := "MachineDB".MachineLimit.Z1Safety.PosMax,
                         MarginSoft := "MachineDB".MachineLimit.Z1Safety.SafetyMargin,
                         MarginHard := "MachineDB".MachineLimit.Z1Safety.SafetyMargin,
                         MotionLock := "WebDB".SystemStatus.DoorSensor,
                         AXISEnabled := "CMMS_Z1_FHPP_CTRL_DB".DriveEnabled,
                         AXISPosOk := "CMMS_Z1_FHPP_CTRL_DB".Ready,
                         AXISReference := "CMMS_Z1_FHPP_CTRL_DB".HomingValid,
                         AXISAxisWarning := "CMMS_Z1_FHPP_CTRL_DB".Warning,
                         AXISAxisError := "CMMS_Z1_FHPP_CTRL_DB".Fault,
                         AXISLockout := "CMMS_Z1_FHPP_CTRL_DB".StandStillControl,
                         AXISActVelocity := "CMMS_Z1_FHPP_CTRL_DB".ActualVelocity,
                         AXISActPosition := "CMMS_Z1_FHPP_CTRL_DB".ActualPosition,
                         AXISAxisAckSetpoint := "CMMS_Z1_FHPP_CTRL_DB".AckStart,
                         AXISReady4Motion := "CMMS_Z1_FHPP_CTRL_DB".Ready,
                         JogStartPos := "MachineDB".MachineLimit.Z1Safety.PosMin,
                         JogEndPos := "MachineDB".MachineLimit.Z1Safety.PosMax,
                         AxisType := 3,
                         YPosition := "WebDB".YOutput.ActualPosition,
                         PositionDelay := "AXES_Positions_Delays".AXIS_Z1_Position_DelayOut,
                         NoGoZoneActive := "WebDB".NoGoZone01Status.NoGoZone01Active,
                         NoGoZoneHomingPermission := "WebDB".NoGoZone01AxisControl.HomingPermissionZ1,
                         NoGoZoneMovePermission := "WebDB".NoGoZone01AxisControl.NoGoMotionLockZ1move,
                         NoGoZoneJogPosPermission := "WebDB".NoGoZone01AxisControl.NoGoMotionLockZ1jog,
                         StartTask := "WebDB".Z1Input.StartTask,
                         Execute := "WebDB".Z1Input.ExecuteFunction,
                         Homing := "WebDB".Z1Input.StartHoming,
                         Status => "WebDB".Z1AddOn1.Error_message_Z1,
                         Overrange => "WebDB".Z1AddOn1.Z1Overrange,
                         Ready => "WebDB".Z1Output.Ready,
                         DriveStop => "WebDB".Z1Output.DriveMoving,
                         Standstill => "WebDB".Z1Output.StandStillControl,
                         MC => "WebDB".Z1Output.MC,
                         AXISEnableAxis => "CMMS_Z1_FHPP_CTRL_DB".EnableDrive,
                         AXISCancelTraversing => "CMMS_Z1_FHPP_CTRL_DB".Halt,
                         AXISIntermediateStop => "CMMS_Z1_FHPP_CTRL_DB".Stop,
                         AXISJog1 => "CMMS_Z1_FHPP_CTRL_DB".JogPos,
                         AXISJog2 => "CMMS_Z1_FHPP_CTRL_DB".JogNeg,
                         AXISAckError => "CMMS_Z1_FHPP_CTRL_DB".ResetFault,
                         AXISExecuteMode => "CMMS_Z1_FHPP_CTRL_DB".StartTask,
                         AXISPosition => "CMMS_Z1_FHPP_CTRL_DB".SetValuePosition,
                         AXISVelocity => "CMMS_Z1_FHPP_CTRL_DB".SetValueVelocity,
                         AXISRelative => "CMMS_Z1_FHPP_CTRL_DB".Relative,
                         AXISHoming => "CMMS_Z1_FHPP_CTRL_DB".StartHoming,
                         FinishTask_Delay => "AXES_Positions_Delays".AXIS_Z1_Position_DelayIn);
   END_IF;
   IF "MachineDB".ArmadilloOption.ZAxisDriveOption = 'CMMS' THEN
       "CMMS_Z1_Movement_DB"();   // "CMMS_Z1_Movement"
   END_IF;
END_REGION

REGION Network 3: AXIZ Z1 Delays
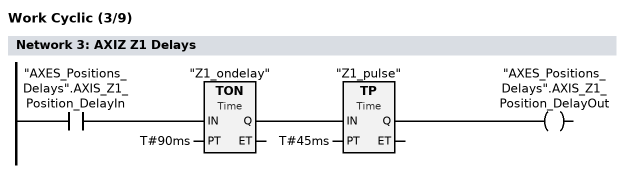
   RUNG wire#powerrail
      Contact( "AXES_Positions_Delays".AXIS_Z1_Position_DelayIn )
      { S7_Templates := "time_type := Time" } "Z1_ondelay".TON(pt := T#90ms, et =>)
      { S7_Templates := "time_type := Time" } "Z1_pulse".TP(pt := T#45ms, et =>)
      Coil( "AXES_Positions_Delays".AXIS_Z1_Position_DelayOut )
   END_RUNG
   // the same network as SCL:
   "Z1_ondelay".TON(IN := "AXES_Positions_Delays".AXIS_Z1_Position_DelayIn, PT := T#90ms);
   "Z1_pulse".TP(IN := "Z1_ondelay".Q, PT := T#45ms);
   "AXES_Positions_Delays".AXIS_Z1_Position_DelayOut := "Z1_pulse".Q;
END_REGION

REGION Network 4: AXIS Z2 Control CMMT V2 To Update
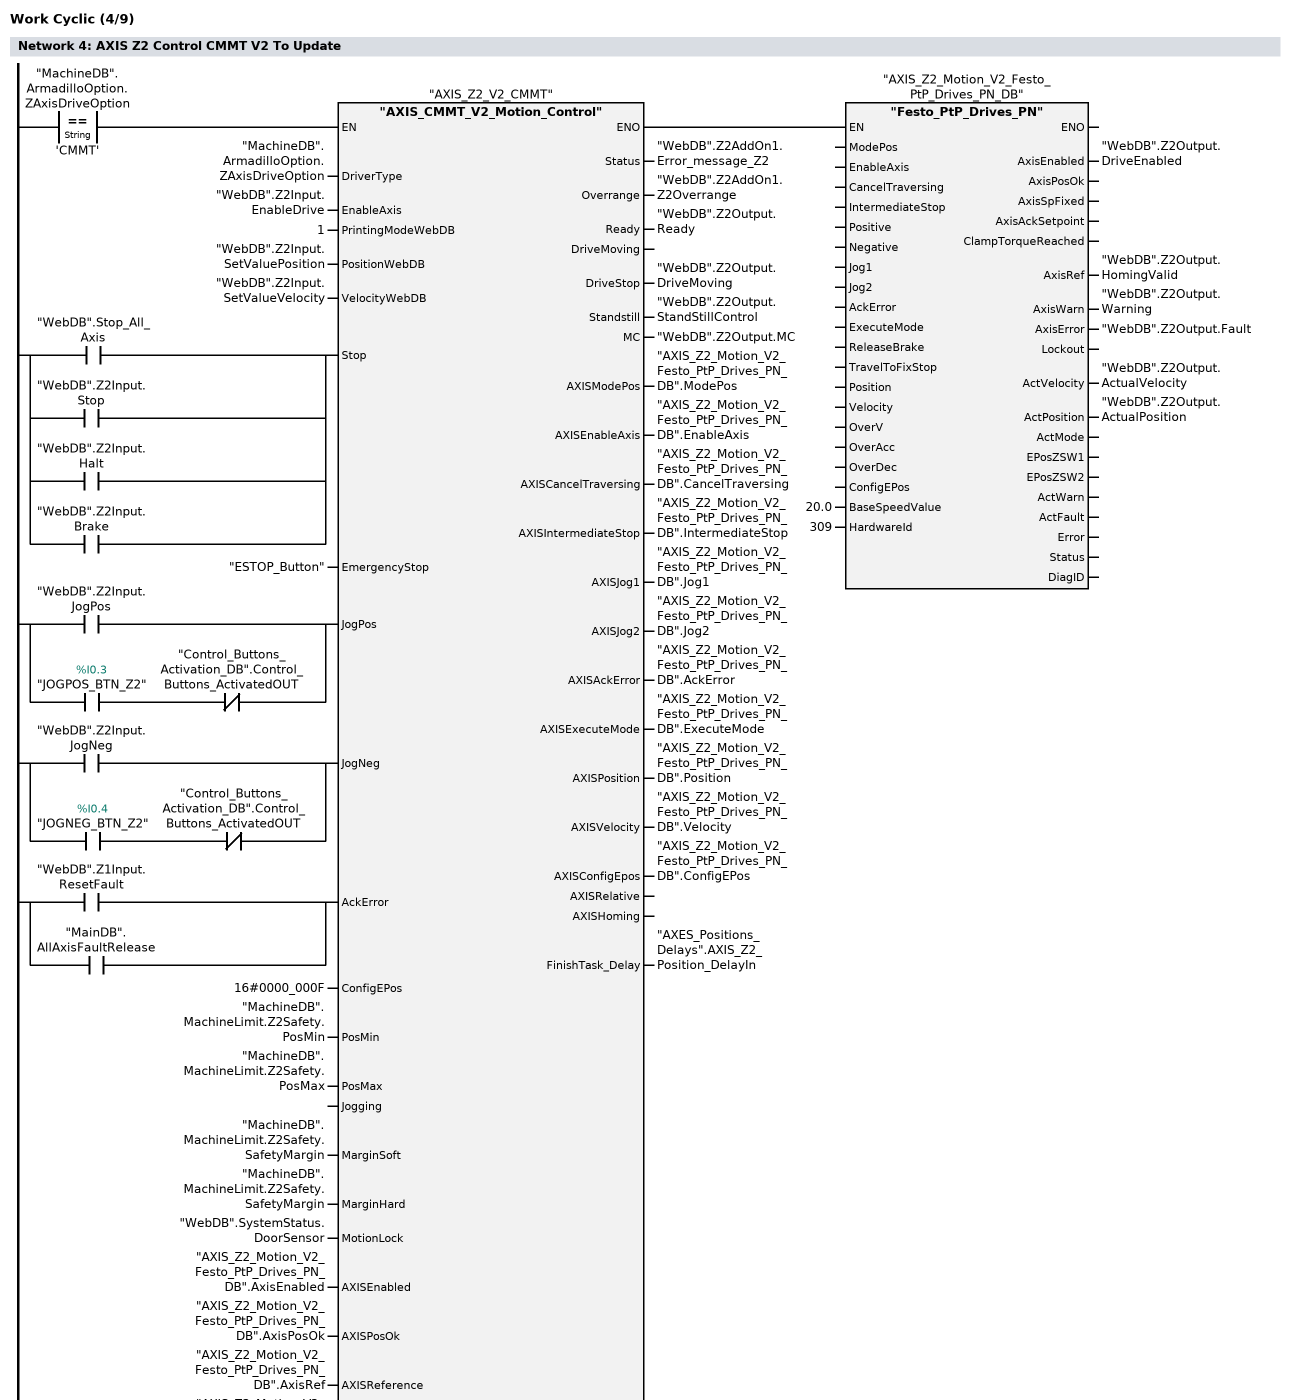
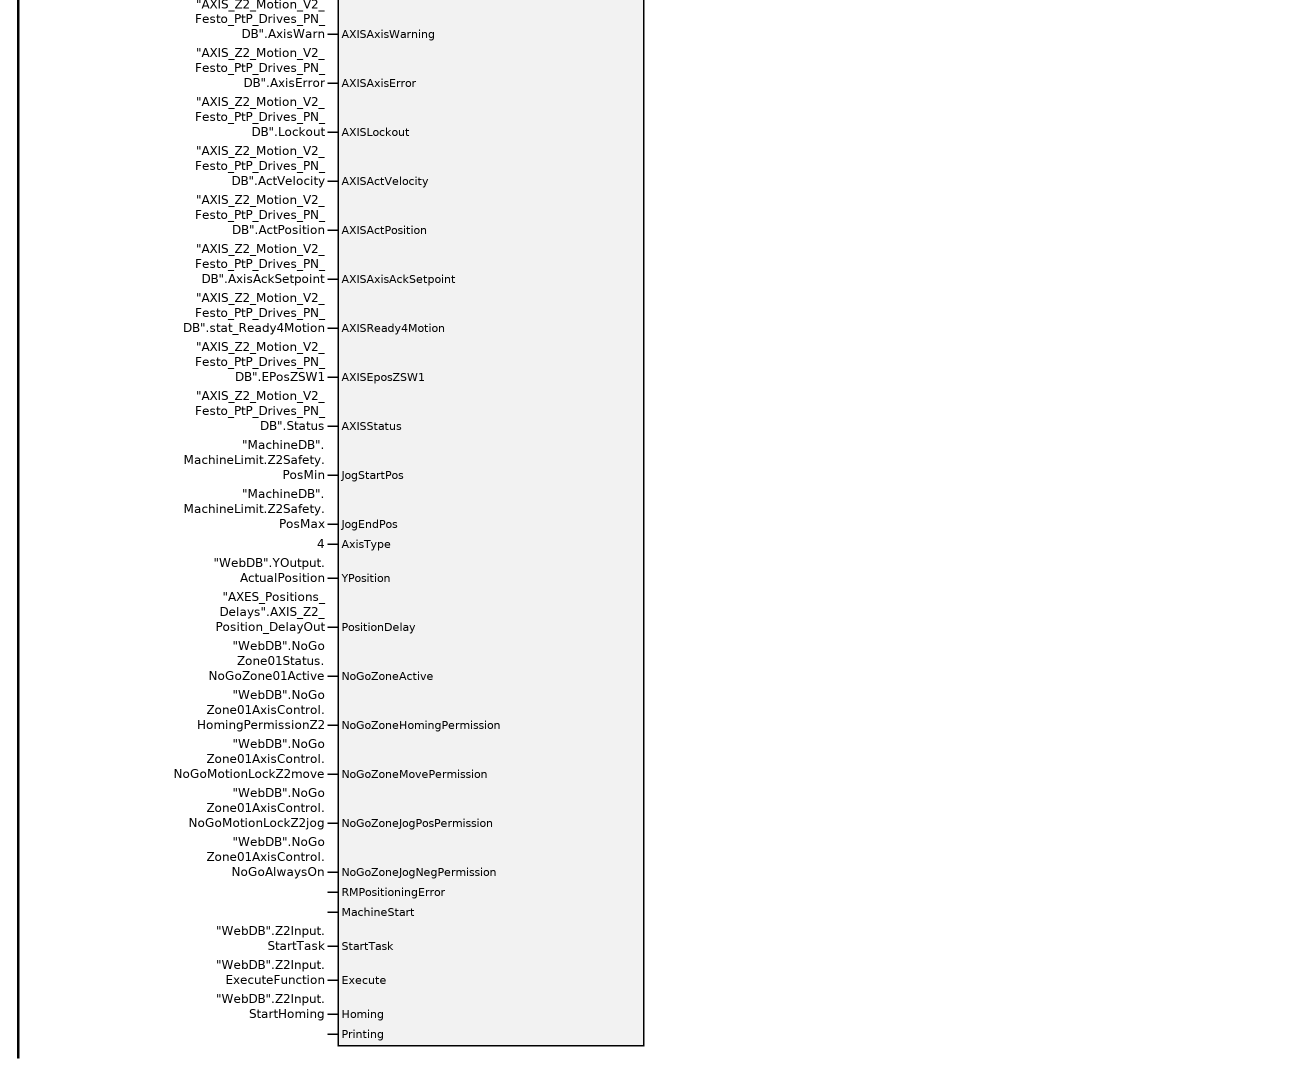
   RUNG wire#powerrail
      { S7_Templates := "SrcType := String" } EQ_Contact(in1 := "MachineDB".ArmadilloOption.ZAxisDriveOption, in2 := 'CMMT')
      "AXIS_Z2_V2_CMMT"(Stop := wire#w1, JogPos := wire#w2, JogNeg := wire#w3, AckError := wire#w4, DriverType := "MachineDB".ArmadilloOption.ZAxisDriveOption, EnableAxis := "WebDB".Z2Input.EnableDrive, PrintingModeWebDB := 1, PositionWebDB := "WebDB".Z2Input.SetValuePosition, VelocityWebDB := "WebDB".Z2Input.SetValueVelocity, EmergencyStop := "ESTOP_Button", ConfigEPos := 16#0000_000F, PosMin := "MachineDB".MachineLimit.Z2Safety.PosMin, PosMax := "MachineDB".MachineLimit.Z2Safety.PosMax, Jogging :=, MarginSoft := "MachineDB".MachineLimit.Z2Safety.SafetyMargin, MarginHard := "MachineDB".MachineLimit.Z2Safety.SafetyMargin, MotionLock := "WebDB".SystemStatus.DoorSensor, AXISEnabled := "AXIS_Z2_Motion_V2_Festo_PtP_Drives_PN_DB".AxisEnabled, AXISPosOk := "AXIS_Z2_Motion_V2_Festo_PtP_Drives_PN_DB".AxisPosOk, AXISReference := "AXIS_Z2_Motion_V2_Festo_PtP_Drives_PN_DB".AxisRef, AXISAxisWarning := "AXIS_Z2_Motion_V2_Festo_PtP_Drives_PN_DB".AxisWarn, AXISAxisError := "AXIS_Z2_Motion_V2_Festo_PtP_Drives_PN_DB".AxisError, AXISLockout := "AXIS_Z2_Motion_V2_Festo_PtP_Drives_PN_DB".Lockout, AXISActVelocity := "AXIS_Z2_Motion_V2_Festo_PtP_Drives_PN_DB".ActVelocity, AXISActPosition := "AXIS_Z2_Motion_V2_Festo_PtP_Drives_PN_DB".ActPosition, AXISAxisAckSetpoint := "AXIS_Z2_Motion_V2_Festo_PtP_Drives_PN_DB".AxisAckSetpoint, AXISReady4Motion := "AXIS_Z2_Motion_V2_Festo_PtP_Drives_PN_DB".stat_Ready4Motion, AXISEposZSW1 := "AXIS_Z2_Motion_V2_Festo_PtP_Drives_PN_DB".EPosZSW1, AXISStatus := "AXIS_Z2_Motion_V2_Festo_PtP_Drives_PN_DB".Status, JogStartPos := "MachineDB".MachineLimit.Z2Safety.PosMin, JogEndPos := "MachineDB".MachineLimit.Z2Safety.PosMax, AxisType := 4, YPosition := "WebDB".YOutput.ActualPosition, PositionDelay := "AXES_Positions_Delays".AXIS_Z2_Position_DelayOut, NoGoZoneActive := "WebDB".NoGoZone01Status.NoGoZone01Active, NoGoZoneHomingPermission := "WebDB".NoGoZone01AxisControl.HomingPermissionZ2, NoGoZoneMovePermission := "WebDB".NoGoZone01AxisControl.NoGoMotionLockZ2move, NoGoZoneJogPosPermission := "WebDB".NoGoZone01AxisControl.NoGoMotionLockZ2jog, NoGoZoneJogNegPermission := "WebDB".NoGoZone01AxisControl.NoGoAlwaysOn, RMPositioningError :=, MachineStart :=, StartTask := "WebDB".Z2Input.StartTask, Execute := "WebDB".Z2Input.ExecuteFunction, Homing := "WebDB".Z2Input.StartHoming, Printing :=, Status => "WebDB".Z2AddOn1.Error_message_Z2, Overrange => "WebDB".Z2AddOn1.Z2Overrange, Ready => "WebDB".Z2Output.Ready, DriveMoving =>, DriveStop => "WebDB".Z2Output.DriveMoving, Standstill => "WebDB".Z2Output.StandStillControl, MC => "WebDB".Z2Output.MC, AXISModePos => "AXIS_Z2_Motion_V2_Festo_PtP_Drives_PN_DB".ModePos, AXISEnableAxis => "AXIS_Z2_Motion_V2_Festo_PtP_Drives_PN_DB".EnableAxis, AXISCancelTraversing => "AXIS_Z2_Motion_V2_Festo_PtP_Drives_PN_DB".CancelTraversing, AXISIntermediateStop => "AXIS_Z2_Motion_V2_Festo_PtP_Drives_PN_DB".IntermediateStop, AXISJog1 => "AXIS_Z2_Motion_V2_Festo_PtP_Drives_PN_DB".Jog1, AXISJog2 => "AXIS_Z2_Motion_V2_Festo_PtP_Drives_PN_DB".Jog2, AXISAckError => "AXIS_Z2_Motion_V2_Festo_PtP_Drives_PN_DB".AckError, AXISExecuteMode => "AXIS_Z2_Motion_V2_Festo_PtP_Drives_PN_DB".ExecuteMode, AXISPosition => "AXIS_Z2_Motion_V2_Festo_PtP_Drives_PN_DB".Position, AXISVelocity => "AXIS_Z2_Motion_V2_Festo_PtP_Drives_PN_DB".Velocity, AXISConfigEpos => "AXIS_Z2_Motion_V2_Festo_PtP_Drives_PN_DB".ConfigEPos, AXISRelative =>, AXISHoming =>, FinishTask_Delay => "AXES_Positions_Delays".AXIS_Z2_Position_DelayIn)
      "AXIS_Z2_Motion_V2_Festo_PtP_Drives_PN_DB"(ModePos :=, EnableAxis :=, CancelTraversing :=, IntermediateStop :=, Positive :=, Negative :=, Jog1 :=, Jog2 :=, AckError :=, ExecuteMode :=, ReleaseBrake :=, TravelToFixStop :=, Position :=, Velocity :=, OverV :=, OverAcc :=, OverDec :=, ConfigEPos :=, BaseSpeedValue := 20.0, HardwareId := 309, AxisEnabled => "WebDB".Z2Output.DriveEnabled, AxisPosOk =>, AxisSpFixed =>, AxisAckSetpoint =>, ClampTorqueReached =>, AxisRef => "WebDB".Z2Output.HomingValid, AxisWarn => "WebDB".Z2Output.Warning, AxisError => "WebDB".Z2Output.Fault, Lockout =>, ActVelocity => "WebDB".Z2Output.ActualVelocity, ActPosition => "WebDB".Z2Output.ActualPosition, ActMode =>, EPosZSW1 =>, EPosZSW2 =>, ActWarn =>, ActFault =>, Error =>, Status =>, DiagID =>)
   END_RUNG
   RUNG wire#powerrail
      Contact( "WebDB".Stop_All_Axis )
   END_RUNG wire#w1
   RUNG wire#powerrail
      Contact( "WebDB".Z2Input.Stop )
   END_RUNG wire#w1
   RUNG wire#powerrail
      Contact( "WebDB".Z2Input.Halt )
   END_RUNG wire#w1
   RUNG wire#powerrail
      Contact( "WebDB".Z2Input.Brake )
   END_RUNG wire#w1
   RUNG wire#powerrail
      Contact( "WebDB".Z2Input.JogPos )
   END_RUNG wire#w2
   RUNG wire#powerrail
      Contact( "JOGPOS_BTN_Z2" )
      I_Contact( "Control_Buttons_Activation_DB".Control_Buttons_ActivatedOUT )
   END_RUNG wire#w2
   RUNG wire#powerrail
      Contact( "WebDB".Z2Input.JogNeg )
   END_RUNG wire#w3
   RUNG wire#powerrail
      Contact( "JOGNEG_BTN_Z2" )
      I_Contact( "Control_Buttons_Activation_DB".Control_Buttons_ActivatedOUT )
   END_RUNG wire#w3
   RUNG wire#powerrail
      Contact( "WebDB".Z1Input.ResetFault )
   END_RUNG wire#w4
   RUNG wire#powerrail
      Contact( "MainDB".AllAxisFaultRelease )
   END_RUNG wire#w4
   // the same network as SCL:
   "AXIS_Z2_V2_CMMT"(EN := "MachineDB".ArmadilloOption.ZAxisDriveOption = 'CMMT',   // "AXIS_CMMT_V2_Motion_Control"
                     DriverType := "MachineDB".ArmadilloOption.ZAxisDriveOption,
                     EnableAxis := "WebDB".Z2Input.EnableDrive,
                     PrintingModeWebDB := 1,
                     PositionWebDB := "WebDB".Z2Input.SetValuePosition,
                     VelocityWebDB := "WebDB".Z2Input.SetValueVelocity,
                     Stop := "WebDB".Stop_All_Axis OR "WebDB".Z2Input.Stop OR "WebDB".Z2Input.Halt OR "WebDB".Z2Input.Brake,
                     EmergencyStop := "ESTOP_Button",
                     JogPos := "WebDB".Z2Input.JogPos OR ("JOGPOS_BTN_Z2" AND NOT "Control_Buttons_Activation_DB".Control_Buttons_ActivatedOUT),
                     JogNeg := "WebDB".Z2Input.JogNeg OR ("JOGNEG_BTN_Z2" AND NOT "Control_Buttons_Activation_DB".Control_Buttons_ActivatedOUT),
                     AckError := "WebDB".Z1Input.ResetFault OR "MainDB".AllAxisFaultRelease,
                     ConfigEPos := 16#0000_000F,
                     PosMin := "MachineDB".MachineLimit.Z2Safety.PosMin,
                     PosMax := "MachineDB".MachineLimit.Z2Safety.PosMax,
                     MarginSoft := "MachineDB".MachineLimit.Z2Safety.SafetyMargin,
                     MarginHard := "MachineDB".MachineLimit.Z2Safety.SafetyMargin,
                     MotionLock := "WebDB".SystemStatus.DoorSensor,
                     AXISEnabled := "AXIS_Z2_Motion_V2_Festo_PtP_Drives_PN_DB".AxisEnabled,
                     AXISPosOk := "AXIS_Z2_Motion_V2_Festo_PtP_Drives_PN_DB".AxisPosOk,
                     AXISReference := "AXIS_Z2_Motion_V2_Festo_PtP_Drives_PN_DB".AxisRef,
                     AXISAxisWarning := "AXIS_Z2_Motion_V2_Festo_PtP_Drives_PN_DB".AxisWarn,
                     AXISAxisError := "AXIS_Z2_Motion_V2_Festo_PtP_Drives_PN_DB".AxisError,
                     AXISLockout := "AXIS_Z2_Motion_V2_Festo_PtP_Drives_PN_DB".Lockout,
                     AXISActVelocity := "AXIS_Z2_Motion_V2_Festo_PtP_Drives_PN_DB".ActVelocity,
                     AXISActPosition := "AXIS_Z2_Motion_V2_Festo_PtP_Drives_PN_DB".ActPosition,
                     AXISAxisAckSetpoint := "AXIS_Z2_Motion_V2_Festo_PtP_Drives_PN_DB".AxisAckSetpoint,
                     AXISReady4Motion := "AXIS_Z2_Motion_V2_Festo_PtP_Drives_PN_DB".stat_Ready4Motion,
                     AXISEposZSW1 := "AXIS_Z2_Motion_V2_Festo_PtP_Drives_PN_DB".EPosZSW1,
                     AXISStatus := "AXIS_Z2_Motion_V2_Festo_PtP_Drives_PN_DB".Status,
                     JogStartPos := "MachineDB".MachineLimit.Z2Safety.PosMin,
                     JogEndPos := "MachineDB".MachineLimit.Z2Safety.PosMax,
                     AxisType := 4,
                     YPosition := "WebDB".YOutput.ActualPosition,
                     PositionDelay := "AXES_Positions_Delays".AXIS_Z2_Position_DelayOut,
                     NoGoZoneActive := "WebDB".NoGoZone01Status.NoGoZone01Active,
                     NoGoZoneHomingPermission := "WebDB".NoGoZone01AxisControl.HomingPermissionZ2,
                     NoGoZoneMovePermission := "WebDB".NoGoZone01AxisControl.NoGoMotionLockZ2move,
                     NoGoZoneJogPosPermission := "WebDB".NoGoZone01AxisControl.NoGoMotionLockZ2jog,
                     NoGoZoneJogNegPermission := "WebDB".NoGoZone01AxisControl.NoGoAlwaysOn,
                     StartTask := "WebDB".Z2Input.StartTask,
                     Execute := "WebDB".Z2Input.ExecuteFunction,
                     Homing := "WebDB".Z2Input.StartHoming,
                     Status => "WebDB".Z2AddOn1.Error_message_Z2,
                     Overrange => "WebDB".Z2AddOn1.Z2Overrange,
                     Ready => "WebDB".Z2Output.Ready,
                     DriveStop => "WebDB".Z2Output.DriveMoving,
                     Standstill => "WebDB".Z2Output.StandStillControl,
                     MC => "WebDB".Z2Output.MC,
                     AXISModePos => "AXIS_Z2_Motion_V2_Festo_PtP_Drives_PN_DB".ModePos,
                     AXISEnableAxis => "AXIS_Z2_Motion_V2_Festo_PtP_Drives_PN_DB".EnableAxis,
                     AXISCancelTraversing => "AXIS_Z2_Motion_V2_Festo_PtP_Drives_PN_DB".CancelTraversing,
                     AXISIntermediateStop => "AXIS_Z2_Motion_V2_Festo_PtP_Drives_PN_DB".IntermediateStop,
                     AXISJog1 => "AXIS_Z2_Motion_V2_Festo_PtP_Drives_PN_DB".Jog1,
                     AXISJog2 => "AXIS_Z2_Motion_V2_Festo_PtP_Drives_PN_DB".Jog2,
                     AXISAckError => "AXIS_Z2_Motion_V2_Festo_PtP_Drives_PN_DB".AckError,
                     AXISExecuteMode => "AXIS_Z2_Motion_V2_Festo_PtP_Drives_PN_DB".ExecuteMode,
                     AXISPosition => "AXIS_Z2_Motion_V2_Festo_PtP_Drives_PN_DB".Position,
                     AXISVelocity => "AXIS_Z2_Motion_V2_Festo_PtP_Drives_PN_DB".Velocity,
                     AXISConfigEpos => "AXIS_Z2_Motion_V2_Festo_PtP_Drives_PN_DB".ConfigEPos,
                     FinishTask_Delay => "AXES_Positions_Delays".AXIS_Z2_Position_DelayIn,
                     ENO => #_w1);
   IF #_w1 THEN
       "AXIS_Z2_Motion_V2_Festo_PtP_Drives_PN_DB"(BaseSpeedValue := 20.0,   // "Festo_PtP_Drives_PN"
                               HardwareId := 309,
                               AxisEnabled => "WebDB".Z2Output.DriveEnabled,
                               AxisRef => "WebDB".Z2Output.HomingValid,
                               AxisWarn => "WebDB".Z2Output.Warning,
                               AxisError => "WebDB".Z2Output.Fault,
                               ActVelocity => "WebDB".Z2Output.ActualVelocity,
                               ActPosition => "WebDB".Z2Output.ActualPosition);
   END_IF;
END_REGION

REGION Network 5: AXIS Z2 CMMS
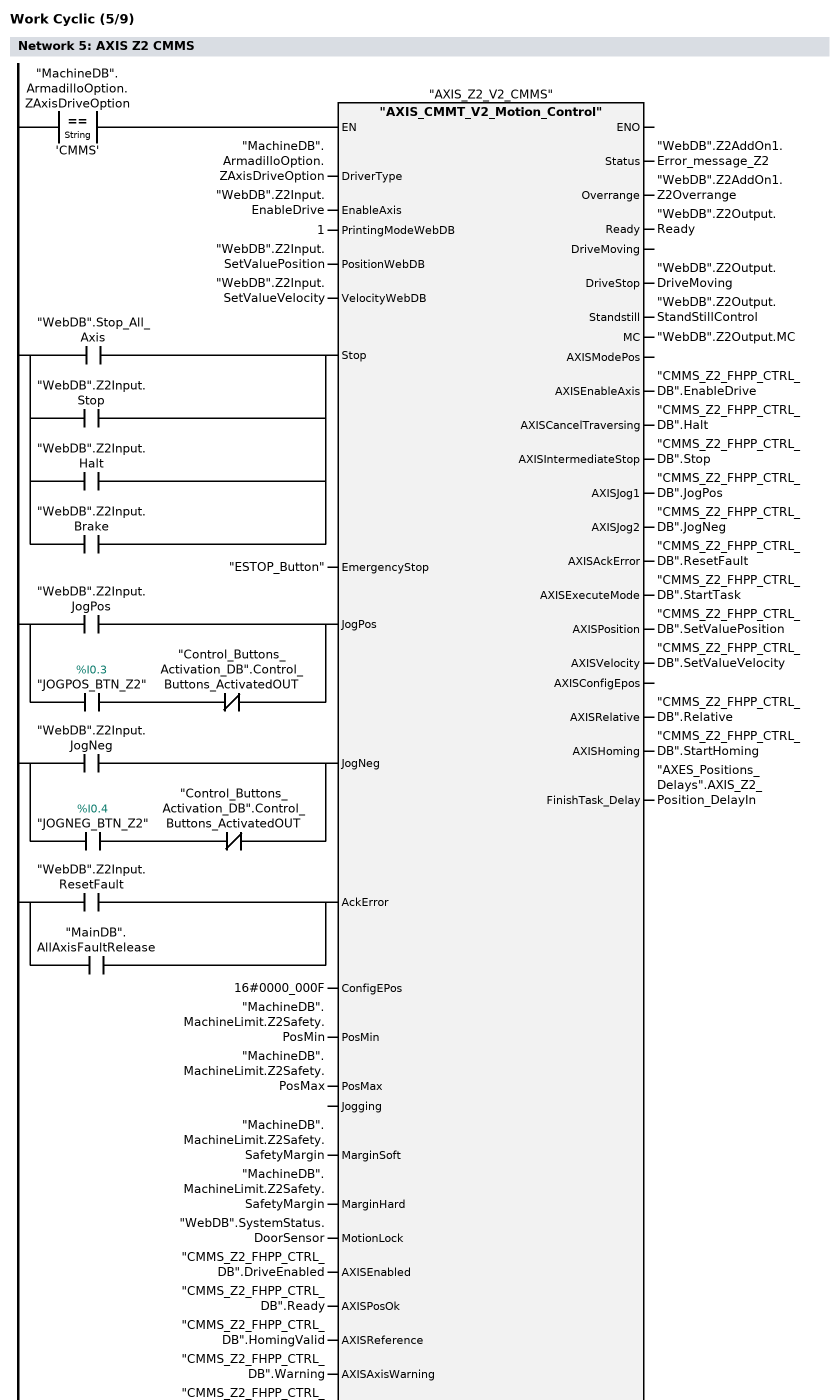
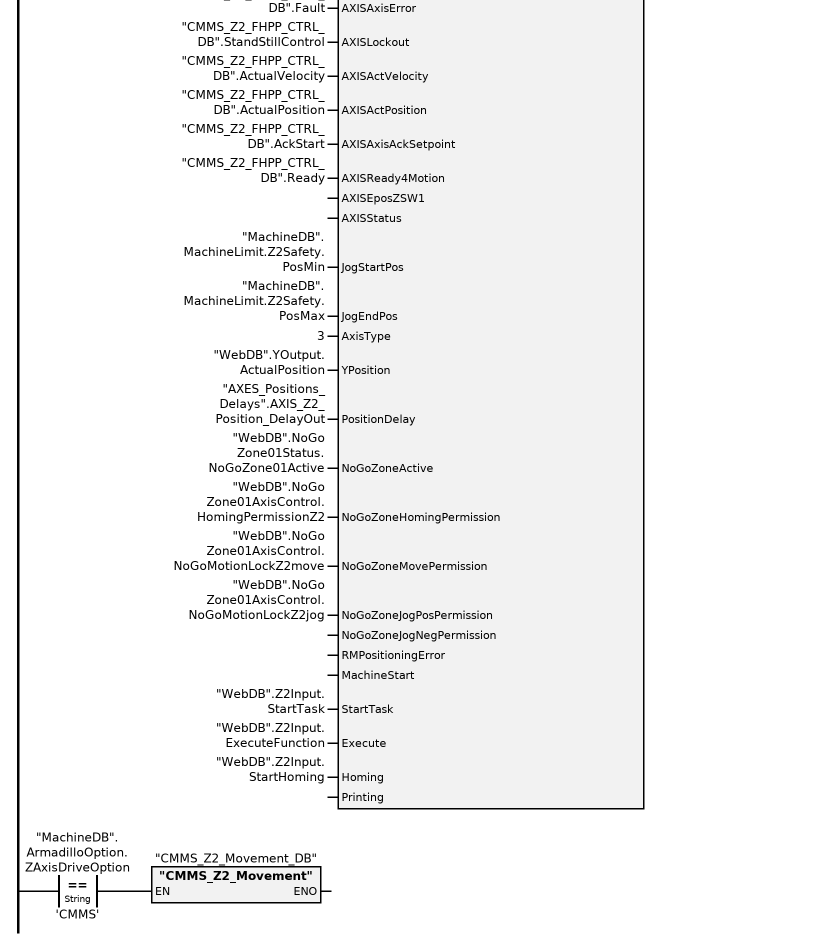
   RUNG wire#powerrail
      { S7_Templates := "SrcType := String" } EQ_Contact(in1 := "MachineDB".ArmadilloOption.ZAxisDriveOption, in2 := 'CMMS')
      "AXIS_Z2_V2_CMMS"(Stop := wire#w1, JogPos := wire#w2, JogNeg := wire#w3, AckError := wire#w4, DriverType := "MachineDB".ArmadilloOption.ZAxisDriveOption, EnableAxis := "WebDB".Z2Input.EnableDrive, PrintingModeWebDB := 1, PositionWebDB := "WebDB".Z2Input.SetValuePosition, VelocityWebDB := "WebDB".Z2Input.SetValueVelocity, EmergencyStop := "ESTOP_Button", ConfigEPos := 16#0000_000F, PosMin := "MachineDB".MachineLimit.Z2Safety.PosMin, PosMax := "MachineDB".MachineLimit.Z2Safety.PosMax, Jogging :=, MarginSoft := "MachineDB".MachineLimit.Z2Safety.SafetyMargin, MarginHard := "MachineDB".MachineLimit.Z2Safety.SafetyMargin, MotionLock := "WebDB".SystemStatus.DoorSensor, AXISEnabled := "CMMS_Z2_FHPP_CTRL_DB".DriveEnabled, AXISPosOk := "CMMS_Z2_FHPP_CTRL_DB".Ready, AXISReference := "CMMS_Z2_FHPP_CTRL_DB".HomingValid, AXISAxisWarning := "CMMS_Z2_FHPP_CTRL_DB".Warning, AXISAxisError := "CMMS_Z2_FHPP_CTRL_DB".Fault, AXISLockout := "CMMS_Z2_FHPP_CTRL_DB".StandStillControl, AXISActVelocity := "CMMS_Z2_FHPP_CTRL_DB".ActualVelocity, AXISActPosition := "CMMS_Z2_FHPP_CTRL_DB".ActualPosition, AXISAxisAckSetpoint := "CMMS_Z2_FHPP_CTRL_DB".AckStart, AXISReady4Motion := "CMMS_Z2_FHPP_CTRL_DB".Ready, AXISEposZSW1 :=, AXISStatus :=, JogStartPos := "MachineDB".MachineLimit.Z2Safety.PosMin, JogEndPos := "MachineDB".MachineLimit.Z2Safety.PosMax, AxisType := 3, YPosition := "WebDB".YOutput.ActualPosition, PositionDelay := "AXES_Positions_Delays".AXIS_Z2_Position_DelayOut, NoGoZoneActive := "WebDB".NoGoZone01Status.NoGoZone01Active, NoGoZoneHomingPermission := "WebDB".NoGoZone01AxisControl.HomingPermissionZ2, NoGoZoneMovePermission := "WebDB".NoGoZone01AxisControl.NoGoMotionLockZ2move, NoGoZoneJogPosPermission := "WebDB".NoGoZone01AxisControl.NoGoMotionLockZ2jog, NoGoZoneJogNegPermission :=, RMPositioningError :=, MachineStart :=, StartTask := "WebDB".Z2Input.StartTask, Execute := "WebDB".Z2Input.ExecuteFunction, Homing := "WebDB".Z2Input.StartHoming, Printing :=, Status => "WebDB".Z2AddOn1.Error_message_Z2, Overrange => "WebDB".Z2AddOn1.Z2Overrange, Ready => "WebDB".Z2Output.Ready, DriveMoving =>, DriveStop => "WebDB".Z2Output.DriveMoving, Standstill => "WebDB".Z2Output.StandStillControl, MC => "WebDB".Z2Output.MC, AXISModePos =>, AXISEnableAxis => "CMMS_Z2_FHPP_CTRL_DB".EnableDrive, AXISCancelTraversing => "CMMS_Z2_FHPP_CTRL_DB".Halt, AXISIntermediateStop => "CMMS_Z2_FHPP_CTRL_DB".Stop, AXISJog1 => "CMMS_Z2_FHPP_CTRL_DB".JogPos, AXISJog2 => "CMMS_Z2_FHPP_CTRL_DB".JogNeg, AXISAckError => "CMMS_Z2_FHPP_CTRL_DB".ResetFault, AXISExecuteMode => "CMMS_Z2_FHPP_CTRL_DB".StartTask, AXISPosition => "CMMS_Z2_FHPP_CTRL_DB".SetValuePosition, AXISVelocity => "CMMS_Z2_FHPP_CTRL_DB".SetValueVelocity, AXISConfigEpos =>, AXISRelative => "CMMS_Z2_FHPP_CTRL_DB".Relative, AXISHoming => "CMMS_Z2_FHPP_CTRL_DB".StartHoming, FinishTask_Delay => "AXES_Positions_Delays".AXIS_Z2_Position_DelayIn)
   END_RUNG
   RUNG wire#powerrail
      Contact( "WebDB".Stop_All_Axis )
   END_RUNG wire#w1
   RUNG wire#powerrail
      Contact( "WebDB".Z2Input.Stop )
   END_RUNG wire#w1
   RUNG wire#powerrail
      Contact( "WebDB".Z2Input.Halt )
   END_RUNG wire#w1
   RUNG wire#powerrail
      Contact( "WebDB".Z2Input.Brake )
   END_RUNG wire#w1
   RUNG wire#powerrail
      Contact( "WebDB".Z2Input.JogPos )
   END_RUNG wire#w2
   RUNG wire#powerrail
      Contact( "JOGPOS_BTN_Z2" )
      I_Contact( "Control_Buttons_Activation_DB".Control_Buttons_ActivatedOUT )
   END_RUNG wire#w2
   RUNG wire#powerrail
      Contact( "WebDB".Z2Input.JogNeg )
   END_RUNG wire#w3
   RUNG wire#powerrail
      Contact( "JOGNEG_BTN_Z2" )
      I_Contact( "Control_Buttons_Activation_DB".Control_Buttons_ActivatedOUT )
   END_RUNG wire#w3
   RUNG wire#powerrail
      Contact( "WebDB".Z2Input.ResetFault )
   END_RUNG wire#w4
   RUNG wire#powerrail
      Contact( "MainDB".AllAxisFaultRelease )
   END_RUNG wire#w4
   RUNG wire#powerrail
      { S7_Templates := "SrcType := String" } EQ_Contact(in1 := "MachineDB".ArmadilloOption.ZAxisDriveOption, in2 := 'CMMS')
      "CMMS_Z2_Movement_DB"()
   END_RUNG
   // the same network as SCL:
   IF "MachineDB".ArmadilloOption.ZAxisDriveOption = 'CMMS' THEN
       "AXIS_Z2_V2_CMMS"(DriverType := "MachineDB".ArmadilloOption.ZAxisDriveOption,   // "AXIS_CMMT_V2_Motion_Control"
                         EnableAxis := "WebDB".Z2Input.EnableDrive,
                         PrintingModeWebDB := 1,
                         PositionWebDB := "WebDB".Z2Input.SetValuePosition,
                         VelocityWebDB := "WebDB".Z2Input.SetValueVelocity,
                         Stop := "WebDB".Stop_All_Axis OR "WebDB".Z2Input.Stop OR "WebDB".Z2Input.Halt OR "WebDB".Z2Input.Brake,
                         EmergencyStop := "ESTOP_Button",
                         JogPos := "WebDB".Z2Input.JogPos OR ("JOGPOS_BTN_Z2" AND NOT "Control_Buttons_Activation_DB".Control_Buttons_ActivatedOUT),
                         JogNeg := "WebDB".Z2Input.JogNeg OR ("JOGNEG_BTN_Z2" AND NOT "Control_Buttons_Activation_DB".Control_Buttons_ActivatedOUT),
                         AckError := "WebDB".Z2Input.ResetFault OR "MainDB".AllAxisFaultRelease,
                         ConfigEPos := 16#0000_000F,
                         PosMin := "MachineDB".MachineLimit.Z2Safety.PosMin,
                         PosMax := "MachineDB".MachineLimit.Z2Safety.PosMax,
                         MarginSoft := "MachineDB".MachineLimit.Z2Safety.SafetyMargin,
                         MarginHard := "MachineDB".MachineLimit.Z2Safety.SafetyMargin,
                         MotionLock := "WebDB".SystemStatus.DoorSensor,
                         AXISEnabled := "CMMS_Z2_FHPP_CTRL_DB".DriveEnabled,
                         AXISPosOk := "CMMS_Z2_FHPP_CTRL_DB".Ready,
                         AXISReference := "CMMS_Z2_FHPP_CTRL_DB".HomingValid,
                         AXISAxisWarning := "CMMS_Z2_FHPP_CTRL_DB".Warning,
                         AXISAxisError := "CMMS_Z2_FHPP_CTRL_DB".Fault,
                         AXISLockout := "CMMS_Z2_FHPP_CTRL_DB".StandStillControl,
                         AXISActVelocity := "CMMS_Z2_FHPP_CTRL_DB".ActualVelocity,
                         AXISActPosition := "CMMS_Z2_FHPP_CTRL_DB".ActualPosition,
                         AXISAxisAckSetpoint := "CMMS_Z2_FHPP_CTRL_DB".AckStart,
                         AXISReady4Motion := "CMMS_Z2_FHPP_CTRL_DB".Ready,
                         JogStartPos := "MachineDB".MachineLimit.Z2Safety.PosMin,
                         JogEndPos := "MachineDB".MachineLimit.Z2Safety.PosMax,
                         AxisType := 3,
                         YPosition := "WebDB".YOutput.ActualPosition,
                         PositionDelay := "AXES_Positions_Delays".AXIS_Z2_Position_DelayOut,
                         NoGoZoneActive := "WebDB".NoGoZone01Status.NoGoZone01Active,
                         NoGoZoneHomingPermission := "WebDB".NoGoZone01AxisControl.HomingPermissionZ2,
                         NoGoZoneMovePermission := "WebDB".NoGoZone01AxisControl.NoGoMotionLockZ2move,
                         NoGoZoneJogPosPermission := "WebDB".NoGoZone01AxisControl.NoGoMotionLockZ2jog,
                         StartTask := "WebDB".Z2Input.StartTask,
                         Execute := "WebDB".Z2Input.ExecuteFunction,
                         Homing := "WebDB".Z2Input.StartHoming,
                         Status => "WebDB".Z2AddOn1.Error_message_Z2,
                         Overrange => "WebDB".Z2AddOn1.Z2Overrange,
                         Ready => "WebDB".Z2Output.Ready,
                         DriveStop => "WebDB".Z2Output.DriveMoving,
                         Standstill => "WebDB".Z2Output.StandStillControl,
                         MC => "WebDB".Z2Output.MC,
                         AXISEnableAxis => "CMMS_Z2_FHPP_CTRL_DB".EnableDrive,
                         AXISCancelTraversing => "CMMS_Z2_FHPP_CTRL_DB".Halt,
                         AXISIntermediateStop => "CMMS_Z2_FHPP_CTRL_DB".Stop,
                         AXISJog1 => "CMMS_Z2_FHPP_CTRL_DB".JogPos,
                         AXISJog2 => "CMMS_Z2_FHPP_CTRL_DB".JogNeg,
                         AXISAckError => "CMMS_Z2_FHPP_CTRL_DB".ResetFault,
                         AXISExecuteMode => "CMMS_Z2_FHPP_CTRL_DB".StartTask,
                         AXISPosition => "CMMS_Z2_FHPP_CTRL_DB".SetValuePosition,
                         AXISVelocity => "CMMS_Z2_FHPP_CTRL_DB".SetValueVelocity,
                         AXISRelative => "CMMS_Z2_FHPP_CTRL_DB".Relative,
                         AXISHoming => "CMMS_Z2_FHPP_CTRL_DB".StartHoming,
                         FinishTask_Delay => "AXES_Positions_Delays".AXIS_Z2_Position_DelayIn);
   END_IF;
   IF "MachineDB".ArmadilloOption.ZAxisDriveOption = 'CMMS' THEN
       "CMMS_Z2_Movement_DB"();   // "CMMS_Z2_Movement"
   END_IF;
END_REGION

REGION Network 6: AXIS Z2 Delays
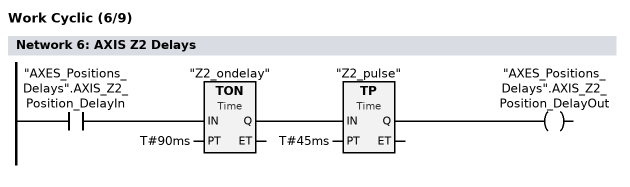
   RUNG wire#powerrail
      Contact( "AXES_Positions_Delays".AXIS_Z2_Position_DelayIn )
      { S7_Templates := "time_type := Time" } "Z2_ondelay".TON(pt := T#90ms, et =>)
      { S7_Templates := "time_type := Time" } "Z2_pulse".TP(pt := T#45ms, et =>)
      Coil( "AXES_Positions_Delays".AXIS_Z2_Position_DelayOut )
   END_RUNG
   // the same network as SCL:
   "Z2_ondelay".TON(IN := "AXES_Positions_Delays".AXIS_Z2_Position_DelayIn, PT := T#90ms);
   "Z2_pulse".TP(IN := "Z2_ondelay".Q, PT := T#45ms);
   "AXES_Positions_Delays".AXIS_Z2_Position_DelayOut := "Z2_pulse".Q;
END_REGION

REGION Network 7: AXIS X Control CMMT V2 To Update
